LIN {X -0.071,Y -649.806,Z 548.445,A 0.000,B 0.000,C 90.000,E1 296.052} C_DIS
LIN {X 0.120,Y -649.563,Z 548.442,A 0.000,B 0.000,C 90.000,E1 295.540} C_DIS
LIN {X 0.217,Y -649.367,Z 548.441,A 0.000,B 0.000,C 90.000,E1 295.283} C_DIS
LIN {X -0.141,Y -646.576,Z 548.437,A 0.000,B 0.000,C 90.000,E1 294.695} C_DIS
LIN {X -0.098,Y -645.526,Z 548.436,A 0.000,B 0.000,C 90.000,E1 294.567} C_DIS
LIN {X -0.323,Y -643.886,Z 548.436,A 0.000,B 0.000,C 90.000,E1 294.463} C_DIS
LIN {X -0.018,Y -639.889,Z 548.434,A 0.000,B 0.000,C 90.000,E1 294.079} C_DIS
LIN {X 0.281,Y -635.567,Z 548.433,A 0.000,B 0.000,C 90.000,E1 293.823} C_DIS
LIN {X -0.032,Y -633.990,Z 548.432,A 0.000,B 0.000,C 90.000,E1 293.770} C_DIS
LIN {X -0.087,Y -632.744,Z 548.432,A 0.000,B 0.000,C 90.000,E1 293.695} C_DIS
LIN {X -0.057,Y -629.987,Z 548.431,A 0.000,B 0.000,C 90.000,E1 293.567} C_DIS
LIN {X -0.135,Y -626.756,Z 548.430,A 0.000,B 0.000,C 90.000,E1 293.462} C_DIS
LIN {X 0.125,Y -623.496,Z 548.429,A 0.000,B 0.000,C 90.000,E1 293.259} C_DIS
LIN {X 0.359,Y -616.119,Z 548.428,A 0.000,B 0.000,C 90.000,E1 292.950} C_DIS
LIN {X -0.008,Y -600.900,Z 548.425,A 0.000,B 0.000,C 90.000,E1 292.461} C_DIS
LIN {X -0.245,Y -582.055,Z 548.421,A 0.000,B 0.000,C 90.000,E1 291.844} C_DIS
LIN {X -0.113,Y -580.503,Z 548.421,A 0.000,B 0.000,C 90.000,E1 291.770} C_DIS
LIN {X 0.230,Y -574.157,Z 548.419,A 0.000,B 0.000,C 90.000,E1 291.408} C_DIS
LIN {X 0.077,Y -570.935,Z 548.418,A 0.000,B 0.000,C 90.000,E1 291.173} C_DIS
LIN {X -0.014,Y -570.080,Z 548.417,A 0.000,B 0.000,C 90.000,E1 291.046} C_DIS
LIN {X -0.057,Y -570.072,Z 548.417,A 0.000,B 0.000,C 90.000,E1 291.046} C_DIS
LIN {X 0.228,Y -569.535,Z 548.414,A 0.000,B 0.000,C 90.000,E1 290.556} C_DIS
LIN {X -0.116,Y -569.520,Z 548.405,A 0.000,B 0.000,C 90.000,E1 288.960} C_DIS
LIN {X -0.023,Y -569.321,Z 548.398,A 0.000,B 0.000,C 90.000,E1 287.583} C_DIS
LIN {X -0.099,Y -569.023,Z 548.392,A 0.000,B 0.000,C 90.000,E1 286.496} C_DIS
LIN {X 0.205,Y -568.590,Z 548.386,A 0.000,B 0.000,C 90.000,E1 285.371} C_DIS
LIN {X 0.131,Y -567.803,Z 548.378,A 0.000,B 0.000,C 90.000,E1 284.008} C_DIS
LIN {X 0.037,Y -567.041,Z 548.370,A 0.000,B 0.000,C 90.000,E1 282.647} C_DIS
LIN {X -0.030,Y -566.172,Z 548.361,A 0.000,B 0.000,C 90.000,E1 281.007} C_DIS
LIN {X -0.149,Y -565.171,Z 548.350,A 0.000,B 0.000,C 90.000,E1 279.095} C_DIS
LIN {X -0.281,Y -564.291,Z 548.340,A 0.000,B 0.000,C 90.000,E1 277.182} C_DIS
LIN {X -0.197,Y -563.753,Z 548.332,A 0.000,B 0.000,C 90.000,E1 275.796} C_DIS
LIN {X -0.082,Y -563.094,Z 548.323,A 0.000,B 0.000,C 90.000,E1 274.131} C_DIS
LIN {X -0.079,Y -562.422,Z 548.315,A 0.000,B 0.000,C 90.000,E1 272.751} C_DIS
LIN {X -0.026,Y -561.613,Z 548.306,A 0.000,B 0.000,C 90.000,E1 271.088} C_DIS
LIN {X 0.096,Y -560.451,Z 548.295,A 0.000,B 0.000,C 90.000,E1 269.141} C_DIS
LIN {X 0.017,Y -559.633,Z 548.288,A 0.000,B 0.000,C 90.000,E1 267.764} C_DIS
LIN {X -0.073,Y -558.784,Z 548.280,A 0.000,B 0.000,C 90.000,E1 266.388} C_DIS
LIN {X 0.055,Y -557.518,Z 548.269,A 0.000,B 0.000,C 90.000,E1 264.432} C_DIS
LIN {X 0.083,Y -556.351,Z 548.260,A 0.000,B 0.000,C 90.000,E1 262.761} C_DIS
LIN {X 0.022,Y -555.263,Z 548.252,A 0.000,B 0.000,C 90.000,E1 261.376} C_DIS
LIN {X -0.141,Y -554.368,Z 548.247,A 0.000,B 0.000,C 90.000,E1 260.557} C_DIS
LIN {X 0.209,Y -551.666,Z 548.235,A 0.000,B 0.000,C 90.000,E1 258.285} C_DIS
LIN {X 0.246,Y -550.027,Z 548.227,A 0.000,B 0.000,C 90.000,E1 256.881} C_DIS
LIN {X -0.156,Y -548.168,Z 548.219,A 0.000,B 0.000,C 90.000,E1 255.519} C_DIS
LIN {X -0.153,Y -546.644,Z 548.213,A 0.000,B 0.000,C 90.000,E1 254.393} C_DIS
LIN {X -0.176,Y -544.912,Z 548.207,A 0.000,B 0.000,C 90.000,E1 253.268} C_DIS
LIN {X -0.291,Y -542.060,Z 548.198,A 0.000,B 0.000,C 90.000,E1 251.583} C_DIS
LIN {X -0.054,Y -540.059,Z 548.191,A 0.000,B 0.000,C 90.000,E1 250.423} C_DIS
LIN {X -0.066,Y -538.426,Z 548.187,A 0.000,B 0.000,C 90.000,E1 249.571} C_DIS
LIN {X -0.167,Y -535.507,Z 548.179,A 0.000,B 0.000,C 90.000,E1 248.156} C_DIS
LIN {X -0.114,Y -532.460,Z 548.171,A 0.000,B 0.000,C 90.000,E1 246.719} C_DIS
LIN {X -0.115,Y -529.083,Z 548.163,A 0.000,B 0.000,C 90.000,E1 245.281} C_DIS
LIN {X 0.113,Y -526.222,Z 548.156,A 0.000,B 0.000,C 90.000,E1 244.101} C_DIS
LIN {X 0.047,Y -523.179,Z 548.150,A 0.000,B 0.000,C 90.000,E1 242.948} C_DIS
LIN {X -0.145,Y -519.278,Z 548.142,A 0.000,B 0.000,C 90.000,E1 241.513} C_DIS
LIN {X 0.298,Y -515.279,Z 548.134,A 0.000,B 0.000,C 90.000,E1 239.999} C_DIS
LIN {X -0.037,Y -512.768,Z 548.129,A 0.000,B 0.000,C 90.000,E1 239.154} C_DIS
LIN {X 0.101,Y -508.301,Z 548.120,A 0.000,B 0.000,C 90.000,E1 237.661} C_DIS
LIN {X 0.156,Y -503.856,Z 548.112,A 0.000,B 0.000,C 90.000,E1 236.167} C_DIS
LIN {X 0.151,Y -497.818,Z 548.101,A 0.000,B 0.000,C 90.000,E1 234.069} C_DIS
LIN {X -0.113,Y -492.012,Z 548.089,A 0.000,B 0.000,C 90.000,E1 231.984} C_DIS
LIN {X -0.087,Y -485.498,Z 548.075,A 0.000,B 0.000,C 90.000,E1 229.542} C_DIS
LIN {X 0.088,Y -480.746,Z 548.065,A 0.000,B 0.000,C 90.000,E1 227.676} C_DIS
LIN {X 0.266,Y -475.303,Z 548.053,A 0.000,B 0.000,C 90.000,E1 225.486} C_DIS
LIN {X -0.044,Y -470.062,Z 548.041,A 0.000,B 0.000,C 90.000,E1 223.338} C_DIS
LIN {X 0.098,Y -465.668,Z 548.030,A 0.000,B 0.000,C 90.000,E1 221.434} C_DIS
LIN {X 0.069,Y -462.782,Z 548.023,A 0.000,B 0.000,C 90.000,E1 220.172} C_DIS
LIN {X 0.133,Y -458.572,Z 548.013,A 0.000,B 0.000,C 90.000,E1 218.257} C_DIS
LIN {X -0.181,Y -454.400,Z 548.002,A 0.000,B 0.000,C 90.000,E1 216.377} C_DIS
LIN {X -0.153,Y -449.717,Z 547.990,A 0.000,B 0.000,C 90.000,E1 214.119} C_DIS
LIN {X 0.166,Y -445.819,Z 547.979,A 0.000,B 0.000,C 90.000,E1 212.133} C_DIS
LIN {X 0.028,Y -440.845,Z 547.964,A 0.000,B 0.000,C 90.000,E1 209.539} C_DIS
LIN {X -0.014,Y -438.499,Z 547.957,A 0.000,B 0.000,C 90.000,E1 208.231} C_DIS
LIN {X -0.039,Y -434.540,Z 547.944,A 0.000,B 0.000,C 90.000,E1 205.924} C_DIS
LIN {X 0.037,Y -430.766,Z 547.931,A 0.000,B 0.000,C 90.000,E1 203.590} C_DIS
LIN {X 0.220,Y -428.218,Z 547.922,A 0.000,B 0.000,C 90.000,E1 201.897} C_DIS
LIN {X 0.005,Y -424.041,Z 547.905,A 0.000,B 0.000,C 90.000,E1 198.906} C_DIS
LIN {X 0.005,Y -420.535,Z 547.890,A 0.000,B 0.000,C 90.000,E1 196.205} C_DIS
LIN {X 0.020,Y -417.754,Z 547.877,A 0.000,B 0.000,C 90.000,E1 193.828} C_DIS
LIN {X -0.077,Y -415.924,Z 547.869,A 0.000,B 0.000,C 90.000,E1 192.479} C_DIS
LIN {X -0.034,Y -413.303,Z 547.858,A 0.000,B 0.000,C 90.000,E1 190.423} C_DIS
LIN {X 0.190,Y -410.163,Z 547.843,A 0.000,B 0.000,C 90.000,E1 187.644} C_DIS
LIN {X -0.181,Y -407.426,Z 547.827,A 0.000,B 0.000,C 90.000,E1 184.935} C_DIS
LIN {X 0.110,Y -404.964,Z 547.812,A 0.000,B 0.000,C 90.000,E1 182.121} C_DIS
LIN {X -0.086,Y -403.054,Z 547.798,A 0.000,B 0.000,C 90.000,E1 179.714} C_DIS
LIN {X 0.111,Y -401.910,Z 547.787,A 0.000,B 0.000,C 90.000,E1 177.593} C_DIS
LIN {X -0.121,Y -400.938,Z 547.773,A 0.000,B 0.000,C 90.000,E1 175.179} C_DIS
LIN {X 0.067,Y -400.447,Z 547.762,A 0.000,B 0.000,C 90.000,E1 173.053} C_DIS
LIN {X -0.095,Y -400.252,Z 547.746,A 0.000,B 0.000,C 90.000,E1 170.274} C_DIS
LIN {X -0.032,Y -400.353,Z 547.732,A 0.000,B 0.000,C 90.000,E1 167.813} C_DIS
LIN {X 0.115,Y -400.928,Z 547.717,A 0.000,B 0.000,C 90.000,E1 164.991} C_DIS
LIN {X 0.022,Y -401.592,Z 547.705,A 0.000,B 0.000,C 90.000,E1 162.906} C_DIS
LIN {X -0.098,Y -402.599,Z 547.692,A 0.000,B 0.000,C 90.000,E1 160.477} C_DIS
LIN {X -0.098,Y -403.321,Z 547.684,A 0.000,B 0.000,C 90.000,E1 159.082} C_DIS
LIN {X 0.117,Y -404.689,Z 547.670,A 0.000,B 0.000,C 90.000,E1 156.613} C_DIS
LIN {X 0.058,Y -405.995,Z 547.659,A 0.000,B 0.000,C 90.000,E1 154.537} C_DIS
LIN {X -0.070,Y -407.105,Z 547.649,A 0.000,B 0.000,C 90.000,E1 152.820} C_DIS
LIN {X 0.202,Y -408.157,Z 547.639,A 0.000,B 0.000,C 90.000,E1 151.051} C_DIS
LIN {X 0.144,Y -409.138,Z 547.630,A 0.000,B 0.000,C 90.000,E1 149.331} C_DIS
LIN {X 0.238,Y -410.037,Z 547.618,A 0.000,B 0.000,C 90.000,E1 147.248} C_DIS
LIN {X 0.227,Y -410.762,Z 547.607,A 0.000,B 0.000,C 90.000,E1 145.182} C_DIS
LIN {X -0.033,Y -411.189,Z 547.597,A 0.000,B 0.000,C 90.000,E1 143.497} C_DIS
LIN {X -0.045,Y -411.527,Z 547.588,A 0.000,B 0.000,C 90.000,E1 141.778} C_DIS
LIN {X -0.022,Y -411.669,Z 547.580,A 0.000,B 0.000,C 90.000,E1 140.400} C_DIS
LIN {X -0.087,Y -411.745,Z 547.570,A 0.000,B 0.000,C 90.000,E1 138.690} C_DIS
LIN {X -0.033,Y -411.839,Z 547.559,A 0.000,B 0.000,C 90.000,E1 136.620} C_DIS
LIN {X 0.146,Y -411.978,Z 547.546,A 0.000,B 0.000,C 90.000,E1 134.190} C_DIS
LIN {X -0.096,Y -412.097,Z 547.534,A 0.000,B 0.000,C 90.000,E1 132.162} C_DIS
LIN {X -0.052,Y -412.028,Z 547.527,A 0.000,B 0.000,C 90.000,E1 130.782} C_DIS
LIN {X 0.135,Y -411.889,Z 547.521,A 0.000,B 0.000,C 90.000,E1 129.725} C_DIS
LIN {X 0.058,Y -411.552,Z 547.515,A 0.000,B 0.000,C 90.000,E1 128.705} C_DIS
LIN {X -0.101,Y -410.959,Z 547.508,A 0.000,B 0.000,C 90.000,E1 127.523} C_DIS
LIN {X -0.139,Y -410.959,Z 547.508,A 0.000,B 0.000,C 90.000,E1 127.523} C_DIS
LIN {X -0.009,Y -415.555,Z 547.500,A 0.000,B 0.000,C 90.000,E1 125.964} C_DIS
LIN {X 0.075,Y -425.946,Z 547.477,A 0.000,B 0.000,C 90.000,E1 121.878} C_DIS
LIN {X 0.029,Y -430.952,Z 547.468,A 0.000,B 0.000,C 90.000,E1 120.207} C_DIS
LIN {X -0.022,Y -440.011,Z 547.448,A 0.000,B 0.000,C 90.000,E1 116.565} C_DIS
LIN {X 0.211,Y -444.409,Z 547.439,A 0.000,B 0.000,C 90.000,E1 115.027} C_DIS
LIN {X 0.170,Y -444.437,Z 547.439,A 0.000,B 0.000,C 90.000,E1 115.027} C_DIS
LIN {X -0.031,Y -463.005,Z 547.435,A 0.000,B 0.000,C 90.000,E1 114.259} C_DIS
LIN {X -0.080,Y -482.164,Z 547.430,A 0.000,B 0.000,C 90.000,E1 113.462} C_DIS
LIN {X 0.029,Y -488.924,Z 547.429,A 0.000,B 0.000,C 90.000,E1 113.153} C_DIS
LIN {X 0.224,Y -495.886,Z 547.427,A 0.000,B 0.000,C 90.000,E1 112.823} C_DIS
LIN {X 0.092,Y -509.292,Z 547.423,A 0.000,B 0.000,C 90.000,E1 112.206} C_DIS
LIN {X -0.001,Y -515.930,Z 547.422,A 0.000,B 0.000,C 90.000,E1 111.897} C_DIS
LIN {X -0.195,Y -522.483,Z 547.420,A 0.000,B 0.000,C 90.000,E1 111.589} C_DIS
LIN {X -0.142,Y -533.967,Z 547.417,A 0.000,B 0.000,C 90.000,E1 110.972} C_DIS
LIN {X -0.109,Y -540.286,Z 547.414,A 0.000,B 0.000,C 90.000,E1 110.610} C_DIS
LIN {X -0.020,Y -547.960,Z 547.412,A 0.000,B 0.000,C 90.000,E1 110.120} C_DIS
LIN {X -0.009,Y -553.960,Z 547.409,A 0.000,B 0.000,C 90.000,E1 109.704} C_DIS
LIN {X -0.265,Y -558.363,Z 547.408,A 0.000,B 0.000,C 90.000,E1 109.396} C_DIS
LIN {X -0.077,Y -563.993,Z 547.405,A 0.000,B 0.000,C 90.000,E1 108.906} C_DIS
LIN {X -0.013,Y -570.154,Z 547.402,A 0.000,B 0.000,C 90.000,E1 108.308} C_DIS
LIN {X 0.142,Y -574.689,Z 547.399,A 0.000,B 0.000,C 90.000,E1 107.819} C_DIS
LIN {X -0.199,Y -577.977,Z 547.397,A 0.000,B 0.000,C 90.000,E1 107.457} C_DIS
LIN {X 0.001,Y -580.308,Z 547.395,A 0.000,B 0.000,C 90.000,E1 107.166} C_DIS
LIN {X 0.297,Y -585.084,Z 547.392,A 0.000,B 0.000,C 90.000,E1 106.496} C_DIS
LIN {X 0.128,Y -589.806,Z 547.388,A 0.000,B 0.000,C 90.000,E1 105.843} C_DIS
LIN {X -0.079,Y -594.976,Z 547.384,A 0.000,B 0.000,C 90.000,E1 105.064} C_DIS
LIN {X -0.099,Y -598.175,Z 547.381,A 0.000,B 0.000,C 90.000,E1 104.537} C_DIS
LIN {X 0.210,Y -602.588,Z 547.376,A 0.000,B 0.000,C 90.000,E1 103.716} C_DIS
LIN {X 0.250,Y -609.039,Z 547.370,A 0.000,B 0.000,C 90.000,E1 102.535} C_DIS
LIN {X 0.085,Y -613.063,Z 547.365,A 0.000,B 0.000,C 90.000,E1 101.771} C_DIS
LIN {X 0.194,Y -615.665,Z 547.363,A 0.000,B 0.000,C 90.000,E1 101.243} C_DIS
LIN {X -0.032,Y -619.092,Z 547.358,A 0.000,B 0.000,C 90.000,E1 100.489} C_DIS
LIN {X -0.117,Y -622.267,Z 547.354,A 0.000,B 0.000,C 90.000,E1 99.726} C_DIS
LIN {X 0.211,Y -628.750,Z 547.346,A 0.000,B 0.000,C 90.000,E1 98.163} C_DIS
LIN {X -0.174,Y -632.914,Z 547.340,A 0.000,B 0.000,C 90.000,E1 97.182} C_DIS
LIN {X -0.071,Y -637.945,Z 547.333,A 0.000,B 0.000,C 90.000,E1 95.910} C_DIS
LIN {X 0.236,Y -641.480,Z 547.327,A 0.000,B 0.000,C 90.000,E1 94.878} C_DIS
LIN {X 0.200,Y -643.859,Z 547.323,A 0.000,B 0.000,C 90.000,E1 94.131} C_DIS
LIN {X -0.044,Y -646.678,Z 547.318,A 0.000,B 0.000,C 90.000,E1 93.154} C_DIS
LIN {X -0.034,Y -648.534,Z 547.313,A 0.000,B 0.000,C 90.000,E1 92.407} C_DIS
LIN {X -0.014,Y -649.948,Z 547.309,A 0.000,B 0.000,C 90.000,E1 91.661} C_DIS
LIN {X 0.000,Y -651.078,Z 547.305,A 0.000,B 0.000,C 90.000,E1 90.917} C_DIS
LIN {X 0.234,Y -651.671,Z 547.302,A 0.000,B 0.000,C 90.000,E1 90.401} C_DIS
LIN {X 0.270,Y -652.305,Z 547.298,A 0.000,B 0.000,C 90.000,E1 89.656} C_DIS
LIN {X 0.309,Y -652.508,Z 547.294,A 0.000,B 0.000,C 90.000,E1 88.912} C_DIS
LIN {X -0.100,Y -652.546,Z 547.291,A 0.000,B 0.000,C 90.000,E1 88.453} C_DIS
LIN {X -0.040,Y -652.236,Z 547.287,A 0.000,B 0.000,C 90.000,E1 87.707} C_DIS
LIN {X -0.009,Y -651.640,Z 547.283,A 0.000,B 0.000,C 90.000,E1 86.963} C_DIS
LIN {X 0.047,Y -650.882,Z 547.279,A 0.000,B 0.000,C 90.000,E1 86.216} C_DIS
LIN {X 0.097,Y -649.758,Z 547.275,A 0.000,B 0.000,C 90.000,E1 85.469} C_DIS
LIN {X -0.029,Y -648.010,Z 547.269,A 0.000,B 0.000,C 90.000,E1 84.489} C_DIS
LIN {X 0.159,Y -647.012,Z 547.267,A 0.000,B 0.000,C 90.000,E1 83.976} C_DIS
LIN {X 0.235,Y -645.175,Z 547.263,A 0.000,B 0.000,C 90.000,E1 83.223} C_DIS
LIN {X 0.302,Y -643.082,Z 547.258,A 0.000,B 0.000,C 90.000,E1 82.470} C_DIS
LIN {X 0.091,Y -639.999,Z 547.253,A 0.000,B 0.000,C 90.000,E1 81.489} C_DIS
LIN {X 0.281,Y -638.350,Z 547.250,A 0.000,B 0.000,C 90.000,E1 80.971} C_DIS
LIN {X 0.097,Y -634.711,Z 547.244,A 0.000,B 0.000,C 90.000,E1 79.982} C_DIS
LIN {X -0.134,Y -630.688,Z 547.239,A 0.000,B 0.000,C 90.000,E1 78.993} C_DIS
LIN {X -0.292,Y -626.257,Z 547.233,A 0.000,B 0.000,C 90.000,E1 77.993} C_DIS
LIN {X 0.106,Y -621.422,Z 547.228,A 0.000,B 0.000,C 90.000,E1 76.937} C_DIS
LIN {X 0.273,Y -618.808,Z 547.225,A 0.000,B 0.000,C 90.000,E1 76.408} C_DIS
LIN {X -0.218,Y -615.267,Z 547.221,A 0.000,B 0.000,C 90.000,E1 75.811} C_DIS
LIN {X -0.290,Y -611.517,Z 547.218,A 0.000,B 0.000,C 90.000,E1 75.172} C_DIS
LIN {X -0.245,Y -607.412,Z 547.214,A 0.000,B 0.000,C 90.000,E1 74.519} C_DIS
LIN {X -0.235,Y -602.951,Z 547.210,A 0.000,B 0.000,C 90.000,E1 73.866} C_DIS
LIN {X -0.094,Y -598.067,Z 547.207,A 0.000,B 0.000,C 90.000,E1 73.196} C_DIS
LIN {X 0.132,Y -594.633,Z 547.204,A 0.000,B 0.000,C 90.000,E1 72.779} C_DIS
LIN {X -0.226,Y -592.933,Z 547.203,A 0.000,B 0.000,C 90.000,E1 72.598} C_DIS
LIN {X -0.060,Y -588.167,Z 547.200,A 0.000,B 0.000,C 90.000,E1 72.054} C_DIS
LIN {X 0.188,Y -583.017,Z 547.197,A 0.000,B 0.000,C 90.000,E1 71.511} C_DIS
LIN {X -0.070,Y -580.127,Z 547.196,A 0.000,B 0.000,C 90.000,E1 71.275} C_DIS
LIN {X 0.274,Y -576.665,Z 547.194,A 0.000,B 0.000,C 90.000,E1 70.913} C_DIS
LIN {X -0.110,Y -571.441,Z 547.192,A 0.000,B 0.000,C 90.000,E1 70.496} C_DIS
LIN {X -0.117,Y -565.989,Z 547.189,A 0.000,B 0.000,C 90.000,E1 70.061} C_DIS
LIN {X -0.106,Y -561.746,Z 547.188,A 0.000,B 0.000,C 90.000,E1 69.752} C_DIS
LIN {X 0.092,Y -555.767,Z 547.185,A 0.000,B 0.000,C 90.000,E1 69.337} C_DIS
LIN {X -0.024,Y -548.840,Z 547.183,A 0.000,B 0.000,C 90.000,E1 68.954} C_DIS
LIN {X 0.168,Y -543.961,Z 547.182,A 0.000,B 0.000,C 90.000,E1 68.666} C_DIS
LIN {X 0.158,Y -536.911,Z 547.180,A 0.000,B 0.000,C 90.000,E1 68.337} C_DIS
LIN {X 0.211,Y -531.587,Z 547.179,A 0.000,B 0.000,C 90.000,E1 68.103} C_DIS
LIN {X -0.037,Y -520.907,Z 547.176,A 0.000,B 0.000,C 90.000,E1 67.720} C_DIS
LIN {X -0.262,Y -513.715,Z 547.175,A 0.000,B 0.000,C 90.000,E1 67.486} C_DIS
LIN {X 0.008,Y -502.871,Z 547.173,A 0.000,B 0.000,C 90.000,E1 67.102} C_DIS
LIN {X -0.116,Y -488.459,Z 547.170,A 0.000,B 0.000,C 90.000,E1 66.666} C_DIS
LIN {X 0.228,Y -462.841,Z 547.166,A 0.000,B 0.000,C 90.000,E1 65.793} C_DIS
LIN {X 0.197,Y -462.827,Z 547.166,A 0.000,B 0.000,C 90.000,E1 65.793} C_DIS
LIN {X 0.180,Y -455.513,Z 547.144,A 0.000,B 0.000,C 90.000,E1 61.897} C_DIS
LIN {X 0.185,Y -445.565,Z 547.119,A 0.000,B 0.000,C 90.000,E1 57.375} C_DIS
LIN {X 0.001,Y -443.781,Z 547.114,A 0.000,B 0.000,C 90.000,E1 56.421} C_DIS
LIN {X -0.160,Y -441.605,Z 547.109,A 0.000,B 0.000,C 90.000,E1 55.595} C_DIS
LIN {X -0.200,Y -441.599,Z 547.109,A 0.000,B 0.000,C 90.000,E1 55.595} C_DIS
LIN {X 0.118,Y -444.210,Z 547.101,A 0.000,B 0.000,C 90.000,E1 54.116} C_DIS
LIN {X -0.138,Y -446.445,Z 547.094,A 0.000,B 0.000,C 90.000,E1 52.844} C_DIS
LIN {X 0.236,Y -449.164,Z 547.084,A 0.000,B 0.000,C 90.000,E1 51.170} C_DIS
LIN {X -0.028,Y -451.203,Z 547.077,A 0.000,B 0.000,C 90.000,E1 49.908} C_DIS
LIN {X -0.259,Y -453.562,Z 547.068,A 0.000,B 0.000,C 90.000,E1 48.324} C_DIS
LIN {X 0.142,Y -455.309,Z 547.061,A 0.000,B 0.000,C 90.000,E1 46.986} C_DIS
LIN {X -0.099,Y -456.400,Z 547.056,A 0.000,B 0.000,C 90.000,E1 46.053} C_DIS
LIN {X -0.011,Y -457.296,Z 547.050,A 0.000,B 0.000,C 90.000,E1 45.081} C_DIS
LIN {X 0.122,Y -458.195,Z 547.043,A 0.000,B 0.000,C 90.000,E1 43.785} C_DIS
LIN {X -0.124,Y -458.624,Z 547.040,A 0.000,B 0.000,C 90.000,E1 43.176} C_DIS
LIN {X 0.019,Y -459.133,Z 547.033,A 0.000,B 0.000,C 90.000,E1 41.881} C_DIS
LIN {X -0.107,Y -459.395,Z 547.026,A 0.000,B 0.000,C 90.000,E1 40.620} C_DIS
LIN {X 0.071,Y -459.405,Z 547.019,A 0.000,B 0.000,C 90.000,E1 39.322} C_DIS
LIN {X 0.050,Y -459.237,Z 547.010,A 0.000,B 0.000,C 90.000,E1 37.729} C_DIS
LIN {X 0.131,Y -458.642,Z 546.999,A 0.000,B 0.000,C 90.000,E1 35.804} C_DIS
LIN {X -0.070,Y -457.878,Z 546.988,A 0.000,B 0.000,C 90.000,E1 33.913} C_DIS
LIN {X -0.053,Y -456.995,Z 546.976,A 0.000,B 0.000,C 90.000,E1 31.671} C_DIS
LIN {X -0.015,Y -456.257,Z 546.965,A 0.000,B 0.000,C 90.000,E1 29.745} C_DIS
LIN {X -0.116,Y -455.310,Z 546.953,A 0.000,B 0.000,C 90.000,E1 27.513} C_DIS
LIN {X -0.047,Y -454.682,Z 546.944,A 0.000,B 0.000,C 90.000,E1 25.899} C_DIS
LIN {X -0.098,Y -453.829,Z 546.930,A 0.000,B 0.000,C 90.000,E1 23.334} C_DIS
LIN {X 0.184,Y -453.283,Z 546.917,A 0.000,B 0.000,C 90.000,E1 21.046} C_DIS
LIN {X 0.025,Y -452.802,Z 546.903,A 0.000,B 0.000,C 90.000,E1 18.489} C_DIS
LIN {X 0.129,Y -452.720,Z 546.888,A 0.000,B 0.000,C 90.000,E1 15.898} C_DIS
LIN {X -0.083,Y -453.063,Z 546.871,A 0.000,B 0.000,C 90.000,E1 12.703} C_DIS
LIN {X -0.217,Y -454.109,Z 546.853,A 0.000,B 0.000,C 90.000,E1 9.500} C_DIS
LIN {X -0.203,Y -455.563,Z 546.837,A 0.000,B 0.000,C 90.000,E1 6.606} C_DIS
LIN {X 0.025,Y -457.200,Z 546.822,A 0.000,B 0.000,C 90.000,E1 4.012} C_DIS
LIN {X 0.201,Y -459.229,Z 546.808,A 0.000,B 0.000,C 90.000,E1 1.432} C_DIS
LIN {X 0.123,Y -461.568,Z 546.795,A 0.000,B 0.000,C 90.000,E1 359.141} C_DIS
LIN {X 0.004,Y -463.826,Z 546.785,A 0.000,B 0.000,C 90.000,E1 357.249} C_DIS
LIN {X 0.214,Y -466.774,Z 546.772,A 0.000,B 0.000,C 90.000,E1 355.008} C_DIS
LIN {X -0.216,Y -468.484,Z 546.765,A 0.000,B 0.000,C 90.000,E1 353.799} C_DIS
LIN {X -0.066,Y -471.004,Z 546.755,A 0.000,B 0.000,C 90.000,E1 351.894} C_DIS
LIN {X 0.168,Y -474.973,Z 546.739,A 0.000,B 0.000,C 90.000,E1 349.050} C_DIS
LIN {X 0.087,Y -478.476,Z 546.727,A 0.000,B 0.000,C 90.000,E1 346.881} C_DIS
LIN {X -0.260,Y -482.194,Z 546.715,A 0.000,B 0.000,C 90.000,E1 344.755} C_DIS
LIN {X 0.083,Y -487.370,Z 546.700,A 0.000,B 0.000,C 90.000,E1 341.945} C_DIS
LIN {X 0.053,Y -490.959,Z 546.690,A 0.000,B 0.000,C 90.000,E1 340.115} C_DIS
LIN {X 0.155,Y -495.167,Z 546.678,A 0.000,B 0.000,C 90.000,E1 337.975} C_DIS
LIN {X 0.019,Y -498.611,Z 546.668,A 0.000,B 0.000,C 90.000,E1 336.177} C_DIS
LIN {X 0.086,Y -501.355,Z 546.659,A 0.000,B 0.000,C 90.000,E1 334.665} C_DIS
LIN {X 0.047,Y -504.590,Z 546.649,A 0.000,B 0.000,C 90.000,E1 332.871} C_DIS
LIN {X -0.079,Y -506.718,Z 546.643,A 0.000,B 0.000,C 90.000,E1 331.691} C_DIS
LIN {X -0.129,Y -510.331,Z 546.631,A 0.000,B 0.000,C 90.000,E1 329.616} C_DIS
LIN {X -0.009,Y -512.971,Z 546.623,A 0.000,B 0.000,C 90.000,E1 328.122} C_DIS
LIN {X -0.264,Y -516.678,Z 546.612,A 0.000,B 0.000,C 90.000,E1 326.087} C_DIS
LIN {X 0.204,Y -519.846,Z 546.602,A 0.000,B 0.000,C 90.000,E1 324.276} C_DIS
LIN {X -0.100,Y -522.978,Z 546.592,A 0.000,B 0.000,C 90.000,E1 322.557} C_DIS
LIN {X -0.050,Y -526.825,Z 546.581,A 0.000,B 0.000,C 90.000,E1 320.517} C_DIS
LIN {X 0.025,Y -530.937,Z 546.569,A 0.000,B 0.000,C 90.000,E1 318.485} C_DIS
LIN {X -0.240,Y -536.135,Z 546.557,A 0.000,B 0.000,C 90.000,E1 316.215} C_DIS
LIN {X 0.019,Y -543.111,Z 546.541,A 0.000,B 0.000,C 90.000,E1 313.338} C_DIS
LIN {X 0.058,Y -546.696,Z 546.533,A 0.000,B 0.000,C 90.000,E1 311.919} C_DIS
LIN {X -0.164,Y -550.764,Z 546.524,A 0.000,B 0.000,C 90.000,E1 310.253} C_DIS
LIN {X 0.299,Y -552.109,Z 546.520,A 0.000,B 0.000,C 90.000,E1 309.644} C_DIS
LIN {X 0.057,Y -554.366,Z 546.516,A 0.000,B 0.000,C 90.000,E1 308.830} C_DIS
LIN {X 0.125,Y -555.260,Z 546.514,A 0.000,B 0.000,C 90.000,E1 308.543} C_DIS
LIN {X 0.198,Y -556.794,Z 546.513,A 0.000,B 0.000,C 90.000,E1 308.257} C_DIS
LIN {X -0.163,Y -558.016,Z 546.511,A 0.000,B 0.000,C 90.000,E1 308.016} C_DIS
LIN {X -0.207,Y -560.843,Z 546.509,A 0.000,B 0.000,C 90.000,E1 307.604} C_DIS
LIN {X 0.009,Y -561.739,Z 546.508,A 0.000,B 0.000,C 90.000,E1 307.443} C_DIS
LIN {X 0.086,Y -565.665,Z 546.506,A 0.000,B 0.000,C 90.000,E1 306.996} C_DIS
LIN {X 0.074,Y -577.991,Z 546.500,A 0.000,B 0.000,C 90.000,E1 305.931} C_DIS
LIN {X 0.214,Y -584.483,Z 546.496,A 0.000,B 0.000,C 90.000,E1 305.311} C_DIS
LIN {X 0.122,Y -588.314,Z 546.494,A 0.000,B 0.000,C 90.000,E1 304.945} C_DIS
LIN {X -0.173,Y -594.560,Z 546.491,A 0.000,B 0.000,C 90.000,E1 304.326} C_DIS
LIN {X 0.013,Y -600.747,Z 546.487,A 0.000,B 0.000,C 90.000,E1 303.658} C_DIS
LIN {X -0.136,Y -610.259,Z 546.481,A 0.000,B 0.000,C 90.000,E1 302.625} C_DIS
LIN {X 0.375,Y -617.069,Z 546.477,A 0.000,B 0.000,C 90.000,E1 301.799} C_DIS
LIN {X 0.102,Y -624.754,Z 546.472,A 0.000,B 0.000,C 90.000,E1 300.924} C_DIS
LIN {X 0.115,Y -629.586,Z 546.468,A 0.000,B 0.000,C 90.000,E1 300.285} C_DIS
LIN {X -0.071,Y -633.038,Z 546.466,A 0.000,B 0.000,C 90.000,E1 299.795} C_DIS
LIN {X 0.019,Y -636.516,Z 546.462,A 0.000,B 0.000,C 90.000,E1 299.155} C_DIS
LIN {X -0.113,Y -639.427,Z 546.459,A 0.000,B 0.000,C 90.000,E1 298.537} C_DIS
LIN {X 0.126,Y -642.898,Z 546.453,A 0.000,B 0.000,C 90.000,E1 297.513} C_DIS
LIN {X 0.267,Y -644.533,Z 546.450,A 0.000,B 0.000,C 90.000,E1 297.001} C_DIS
LIN {X -0.158,Y -645.835,Z 546.447,A 0.000,B 0.000,C 90.000,E1 296.539} C_DIS
LIN {X -0.080,Y -646.463,Z 546.446,A 0.000,B 0.000,C 90.000,E1 296.283} C_DIS
LIN {X 0.002,Y -646.755,Z 546.445,A 0.000,B 0.000,C 90.000,E1 296.027} C_DIS
LIN {X -0.111,Y -646.598,Z 546.442,A 0.000,B 0.000,C 90.000,E1 295.540} C_DIS
LIN {X -0.026,Y -646.074,Z 546.440,A 0.000,B 0.000,C 90.000,E1 295.283} C_DIS
LIN {X 0.140,Y -644.044,Z 546.438,A 0.000,B 0.000,C 90.000,E1 294.771} C_DIS
LIN {X 0.251,Y -640.832,Z 546.436,A 0.000,B 0.000,C 90.000,E1 294.387} C_DIS
LIN {X 0.065,Y -638.226,Z 546.434,A 0.000,B 0.000,C 90.000,E1 294.155} C_DIS
LIN {X 0.108,Y -635.689,Z 546.434,A 0.000,B 0.000,C 90.000,E1 294.027} C_DIS
LIN {X -0.231,Y -632.967,Z 546.433,A 0.000,B 0.000,C 90.000,E1 293.898} C_DIS
LIN {X 0.102,Y -632.502,Z 546.432,A 0.000,B 0.000,C 90.000,E1 293.823} C_DIS
LIN {X 0.160,Y -630.798,Z 546.432,A 0.000,B 0.000,C 90.000,E1 293.695} C_DIS
LIN {X -0.034,Y -627.696,Z 546.431,A 0.000,B 0.000,C 90.000,E1 293.590} C_DIS
LIN {X -0.110,Y -624.102,Z 546.430,A 0.000,B 0.000,C 90.000,E1 293.387} C_DIS
LIN {X 0.297,Y -622.357,Z 546.429,A 0.000,B 0.000,C 90.000,E1 293.259} C_DIS
LIN {X 0.242,Y -612.951,Z 546.427,A 0.000,B 0.000,C 90.000,E1 292.898} C_DIS
LIN {X 0.273,Y -600.603,Z 546.425,A 0.000,B 0.000,C 90.000,E1 292.461} C_DIS
LIN {X -0.003,Y -581.868,Z 546.421,A 0.000,B 0.000,C 90.000,E1 291.844} C_DIS
LIN {X 0.094,Y -576.724,Z 546.420,A 0.000,B 0.000,C 90.000,E1 291.589} C_DIS
LIN {X -0.191,Y -575.181,Z 546.420,A 0.000,B 0.000,C 90.000,E1 291.535} C_DIS
LIN {X 0.229,Y -571.555,Z 546.418,A 0.000,B 0.000,C 90.000,E1 291.227} C_DIS
LIN {X -0.202,Y -571.095,Z 546.418,A 0.000,B 0.000,C 90.000,E1 291.227} C_DIS
LIN {X -0.222,Y -570.643,Z 546.417,A 0.000,B 0.000,C 90.000,E1 291.099} C_DIS
LIN {X -0.252,Y -570.029,Z 546.414,A 0.000,B 0.000,C 90.000,E1 290.556} C_DIS
LIN {X 0.224,Y -570.059,Z 546.406,A 0.000,B 0.000,C 90.000,E1 289.141} C_DIS
LIN {X -0.217,Y -569.904,Z 546.399,A 0.000,B 0.000,C 90.000,E1 287.819} C_DIS
LIN {X -0.114,Y -569.570,Z 546.391,A 0.000,B 0.000,C 90.000,E1 286.441} C_DIS
LIN {X 0.202,Y -569.142,Z 546.385,A 0.000,B 0.000,C 90.000,E1 285.315} C_DIS
LIN {X -0.097,Y -568.179,Z 546.376,A 0.000,B 0.000,C 90.000,E1 283.703} C_DIS
LIN {X 0.059,Y -567.594,Z 546.370,A 0.000,B 0.000,C 90.000,E1 282.591} C_DIS
LIN {X -0.167,Y -566.890,Z 546.362,A 0.000,B 0.000,C 90.000,E1 281.243} C_DIS
LIN {X -0.131,Y -566.283,Z 546.356,A 0.000,B 0.000,C 90.000,E1 280.141} C_DIS
LIN {X 0.244,Y -565.481,Z 546.347,A 0.000,B 0.000,C 90.000,E1 278.454} C_DIS
LIN {X 0.043,Y -564.633,Z 546.336,A 0.000,B 0.000,C 90.000,E1 276.549} C_DIS
LIN {X 0.134,Y -564.109,Z 546.329,A 0.000,B 0.000,C 90.000,E1 275.163} C_DIS
LIN {X 0.154,Y -563.542,Z 546.321,A 0.000,B 0.000,C 90.000,E1 273.784} C_DIS
LIN {X -0.227,Y -562.558,Z 546.310,A 0.000,B 0.000,C 90.000,E1 271.892} C_DIS
LIN {X -0.267,Y -561.784,Z 546.303,A 0.000,B 0.000,C 90.000,E1 270.516} C_DIS
LIN {X -0.142,Y -560.628,Z 546.292,A 0.000,B 0.000,C 90.000,E1 268.568} C_DIS
LIN {X -0.132,Y -559.591,Z 546.283,A 0.000,B 0.000,C 90.000,E1 266.906} C_DIS
LIN {X 0.009,Y -558.286,Z 546.272,A 0.000,B 0.000,C 90.000,E1 264.951} C_DIS
LIN {X -0.143,Y -557.528,Z 546.266,A 0.000,B 0.000,C 90.000,E1 263.856} C_DIS
LIN {X -0.175,Y -556.555,Z 546.258,A 0.000,B 0.000,C 90.000,E1 262.470} C_DIS
LIN {X 0.190,Y -555.683,Z 546.252,A 0.000,B 0.000,C 90.000,E1 261.319} C_DIS
LIN {X 0.031,Y -554.773,Z 546.247,A 0.000,B 0.000,C 90.000,E1 260.500} C_DIS
LIN {X -0.153,Y -552.036,Z 546.235,A 0.000,B 0.000,C 90.000,E1 258.285} C_DIS
LIN {X -0.108,Y -550.358,Z 546.227,A 0.000,B 0.000,C 90.000,E1 256.881} C_DIS
LIN {X 0.027,Y -548.467,Z 546.219,A 0.000,B 0.000,C 90.000,E1 255.463} C_DIS
LIN {X 0.122,Y -546.498,Z 546.211,A 0.000,B 0.000,C 90.000,E1 254.047} C_DIS
LIN {X 0.245,Y -544.701,Z 546.205,A 0.000,B 0.000,C 90.000,E1 252.906} C_DIS
LIN {X 0.124,Y -541.782,Z 546.196,A 0.000,B 0.000,C 90.000,E1 251.221} C_DIS
LIN {X -0.109,Y -539.164,Z 546.188,A 0.000,B 0.000,C 90.000,E1 249.826} C_DIS
LIN {X -0.204,Y -536.260,Z 546.180,A 0.000,B 0.000,C 90.000,E1 248.411} C_DIS
LIN {X -0.143,Y -533.178,Z 546.172,A 0.000,B 0.000,C 90.000,E1 246.975} C_DIS
LIN {X 0.161,Y -530.550,Z 546.166,A 0.000,B 0.000,C 90.000,E1 245.793} C_DIS
LIN {X -0.066,Y -527.701,Z 546.159,A 0.000,B 0.000,C 90.000,E1 244.665} C_DIS
LIN {X -0.106,Y -524.757,Z 546.153,A 0.000,B 0.000,C 90.000,E1 243.512} C_DIS
LIN {X -0.188,Y -521.659,Z 546.146,A 0.000,B 0.000,C 90.000,E1 242.359} C_DIS
LIN {X -0.032,Y -516.875,Z 546.137,A 0.000,B 0.000,C 90.000,E1 240.589} C_DIS
LIN {X 0.011,Y -513.611,Z 546.130,A 0.000,B 0.000,C 90.000,E1 239.410} C_DIS
LIN {X 0.168,Y -509.165,Z 546.122,A 0.000,B 0.000,C 90.000,E1 237.916} C_DIS
LIN {X 0.246,Y -504.720,Z 546.114,A 0.000,B 0.000,C 90.000,E1 236.421} C_DIS
LIN {X -0.181,Y -500.344,Z 546.105,A 0.000,B 0.000,C 90.000,E1 234.975} C_DIS
LIN {X 0.022,Y -494.431,Z 546.094,A 0.000,B 0.000,C 90.000,E1 232.844} C_DIS
LIN {X 0.137,Y -491.133,Z 546.087,A 0.000,B 0.000,C 90.000,E1 231.618} C_DIS
LIN {X -0.060,Y -485.441,Z 546.075,A 0.000,B 0.000,C 90.000,E1 229.504} C_DIS
LIN {X 0.156,Y -480.674,Z 546.065,A 0.000,B 0.000,C 90.000,E1 227.634} C_DIS
LIN {X -0.021,Y -475.224,Z 546.053,A 0.000,B 0.000,C 90.000,E1 225.486} C_DIS
LIN {X -0.094,Y -470.724,Z 546.042,A 0.000,B 0.000,C 90.000,E1 223.623} C_DIS
LIN {X 0.163,Y -465.588,Z 546.030,A 0.000,B 0.000,C 90.000,E1 221.391} C_DIS
LIN {X 0.188,Y -461.965,Z 546.021,A 0.000,B 0.000,C 90.000,E1 219.806} C_DIS
LIN {X 0.110,Y -459.190,Z 546.014,A 0.000,B 0.000,C 90.000,E1 218.543} C_DIS
LIN {X -0.193,Y -454.993,Z 546.004,A 0.000,B 0.000,C 90.000,E1 216.664} C_DIS
LIN {X -0.145,Y -450.293,Z 545.991,A 0.000,B 0.000,C 90.000,E1 214.405} C_DIS
LIN {X 0.192,Y -446.368,Z 545.980,A 0.000,B 0.000,C 90.000,E1 212.418} C_DIS
LIN {X 0.080,Y -441.380,Z 545.966,A 0.000,B 0.000,C 90.000,E1 209.823} C_DIS
LIN {X 0.091,Y -438.420,Z 545.957,A 0.000,B 0.000,C 90.000,E1 208.180} C_DIS
LIN {X -0.143,Y -435.025,Z 545.946,A 0.000,B 0.000,C 90.000,E1 206.232} C_DIS
LIN {X -0.059,Y -431.198,Z 545.933,A 0.000,B 0.000,C 90.000,E1 203.898} C_DIS
LIN {X -0.060,Y -428.134,Z 545.922,A 0.000,B 0.000,C 90.000,E1 201.897} C_DIS
LIN {X 0.126,Y -423.947,Z 545.905,A 0.000,B 0.000,C 90.000,E1 198.852} C_DIS
LIN {X 0.073,Y -420.894,Z 545.892,A 0.000,B 0.000,C 90.000,E1 196.496} C_DIS
LIN {X 0.092,Y -418.086,Z 545.879,A 0.000,B 0.000,C 90.000,E1 194.120} C_DIS
LIN {X -0.003,Y -416.319,Z 545.871,A 0.000,B 0.000,C 90.000,E1 192.771} C_DIS
LIN {X 0.050,Y -413.705,Z 545.860,A 0.000,B 0.000,C 90.000,E1 190.715} C_DIS
LIN {X -0.118,Y -410.537,Z 545.844,A 0.000,B 0.000,C 90.000,E1 187.992} C_DIS
LIN {X -0.028,Y -407.738,Z 545.829,A 0.000,B 0.000,C 90.000,E1 185.220} C_DIS
LIN {X -0.113,Y -405.551,Z 545.816,A 0.000,B 0.000,C 90.000,E1 182.808} C_DIS
LIN {X 0.109,Y -403.624,Z 545.802,A 0.000,B 0.000,C 90.000,E1 180.344} C_DIS
LIN {X -0.120,Y -402.160,Z 545.789,A 0.000,B 0.000,C 90.000,E1 177.936} C_DIS
LIN {X 0.012,Y -401.015,Z 545.773,A 0.000,B 0.000,C 90.000,E1 175.122} C_DIS
LIN {X 0.174,Y -400.464,Z 545.757,A 0.000,B 0.000,C 90.000,E1 172.299} C_DIS
LIN {X 0.096,Y -400.333,Z 545.744,A 0.000,B 0.000,C 90.000,E1 169.859} C_DIS
LIN {X 0.102,Y -400.478,Z 545.732,A 0.000,B 0.000,C 90.000,E1 167.757} C_DIS
LIN {X -0.139,Y -401.062,Z 545.717,A 0.000,B 0.000,C 90.000,E1 164.991} C_DIS
LIN {X -0.230,Y -401.723,Z 545.705,A 0.000,B 0.000,C 90.000,E1 162.906} C_DIS
LIN {X 0.034,Y -402.766,Z 545.691,A 0.000,B 0.000,C 90.000,E1 160.423} C_DIS
LIN {X 0.128,Y -403.697,Z 545.682,A 0.000,B 0.000,C 90.000,E1 158.666} C_DIS
LIN {X 0.132,Y -405.059,Z 545.668,A 0.000,B 0.000,C 90.000,E1 156.230} C_DIS
LIN {X -0.180,Y -406.193,Z 545.658,A 0.000,B 0.000,C 90.000,E1 154.537} C_DIS
LIN {X 0.154,Y -407.545,Z 545.647,A 0.000,B 0.000,C 90.000,E1 152.410} C_DIS
LIN {X 0.161,Y -408.801,Z 545.635,A 0.000,B 0.000,C 90.000,E1 150.333} C_DIS
LIN {X -0.161,Y -409.516,Z 545.628,A 0.000,B 0.000,C 90.000,E1 148.997} C_DIS
LIN {X 0.017,Y -410.261,Z 545.618,A 0.000,B 0.000,C 90.000,E1 147.248} C_DIS
LIN {X 0.090,Y -410.894,Z 545.609,A 0.000,B 0.000,C 90.000,E1 145.515} C_DIS
LIN {X 0.010,Y -411.305,Z 545.601,A 0.000,B 0.000,C 90.000,E1 144.149} C_DIS
LIN {X -0.002,Y -411.660,Z 545.591,A 0.000,B 0.000,C 90.000,E1 142.431} C_DIS
LIN {X 0.080,Y -411.889,Z 545.584,A 0.000,B 0.000,C 90.000,E1 141.045} C_DIS
LIN {X 0.112,Y -411.990,Z 545.576,A 0.000,B 0.000,C 90.000,E1 139.666} C_DIS
LIN {X 0.045,Y -412.075,Z 545.567,A 0.000,B 0.000,C 90.000,E1 137.957} C_DIS
LIN {X 0.220,Y -412.130,Z 545.557,A 0.000,B 0.000,C 90.000,E1 136.215} C_DIS
LIN {X -0.033,Y -412.247,Z 545.546,A 0.000,B 0.000,C 90.000,E1 134.190} C_DIS
LIN {X 0.007,Y -412.374,Z 545.534,A 0.000,B 0.000,C 90.000,E1 132.123} C_DIS
LIN {X 0.049,Y -412.291,Z 545.526,A 0.000,B 0.000,C 90.000,E1 130.744} C_DIS
LIN {X -0.031,Y -412.106,Z 545.521,A 0.000,B 0.000,C 90.000,E1 129.725} C_DIS
LIN {X 0.063,Y -411.565,Z 545.513,A 0.000,B 0.000,C 90.000,E1 128.338} C_DIS
LIN {X 0.085,Y -411.109,Z 545.508,A 0.000,B 0.000,C 90.000,E1 127.443} C_DIS
LIN {X 0.045,Y -411.114,Z 545.508,A 0.000,B 0.000,C 90.000,E1 127.443} C_DIS
LIN {X 0.076,Y -415.617,Z 545.500,A 0.000,B 0.000,C 90.000,E1 125.931} C_DIS
LIN {X -0.065,Y -425.048,Z 545.479,A 0.000,B 0.000,C 90.000,E1 122.212} C_DIS
LIN {X -0.134,Y -431.000,Z 545.468,A 0.000,B 0.000,C 90.000,E1 120.207} C_DIS
LIN {X 0.012,Y -440.071,Z 545.448,A 0.000,B 0.000,C 90.000,E1 116.539} C_DIS
LIN {X 0.009,Y -444.853,Z 545.438,A 0.000,B 0.000,C 90.000,E1 114.899} C_DIS
LIN {X -0.106,Y -445.155,Z 545.438,A 0.000,B 0.000,C 90.000,E1 114.771} C_DIS
LIN {X -0.146,Y -445.182,Z 545.438,A 0.000,B 0.000,C 90.000,E1 114.771} C_DIS
LIN {X 0.126,Y -466.749,Z 545.432,A 0.000,B 0.000,C 90.000,E1 113.823} C_DIS
LIN {X -0.107,Y -484.163,Z 545.428,A 0.000,B 0.000,C 90.000,E1 113.131} C_DIS
LIN {X 0.248,Y -494.383,Z 545.426,A 0.000,B 0.000,C 90.000,E1 112.642} C_DIS
LIN {X 0.269,Y -501.136,Z 545.424,A 0.000,B 0.000,C 90.000,E1 112.333} C_DIS
LIN {X 0.162,Y -514.532,Z 545.421,A 0.000,B 0.000,C 90.000,E1 111.716} C_DIS
LIN {X 0.035,Y -521.220,Z 545.419,A 0.000,B 0.000,C 90.000,E1 111.408} C_DIS
LIN {X 0.237,Y -532.641,Z 545.416,A 0.000,B 0.000,C 90.000,E1 110.791} C_DIS
LIN {X -0.027,Y -540.676,Z 545.413,A 0.000,B 0.000,C 90.000,E1 110.375} C_DIS
LIN {X -0.004,Y -546.889,Z 545.411,A 0.000,B 0.000,C 90.000,E1 109.993} C_DIS
LIN {X 0.138,Y -552.897,Z 545.409,A 0.000,B 0.000,C 90.000,E1 109.577} C_DIS
LIN {X 0.064,Y -557.207,Z 545.407,A 0.000,B 0.000,C 90.000,E1 109.268} C_DIS
LIN {X -0.080,Y -564.019,Z 545.404,A 0.000,B 0.000,C 90.000,E1 108.725} C_DIS
LIN {X -0.063,Y -569.293,Z 545.401,A 0.000,B 0.000,C 90.000,E1 108.236} C_DIS
LIN {X 0.262,Y -574.323,Z 545.398,A 0.000,B 0.000,C 90.000,E1 107.692} C_DIS
LIN {X 0.205,Y -579.029,Z 545.396,A 0.000,B 0.000,C 90.000,E1 107.166} C_DIS
LIN {X -0.090,Y -585.281,Z 545.391,A 0.000,B 0.000,C 90.000,E1 106.386} C_DIS
LIN {X -0.097,Y -590.056,Z 545.387,A 0.000,B 0.000,C 90.000,E1 105.717} C_DIS
LIN {X -0.231,Y -594.490,Z 545.384,A 0.000,B 0.000,C 90.000,E1 105.064} C_DIS
LIN {X -0.255,Y -597.783,Z 545.381,A 0.000,B 0.000,C 90.000,E1 104.537} C_DIS
LIN {X 0.049,Y -602.349,Z 545.376,A 0.000,B 0.000,C 90.000,E1 103.716} C_DIS
LIN {X -0.245,Y -607.478,Z 545.371,A 0.000,B 0.000,C 90.000,E1 102.827} C_DIS
LIN {X -0.128,Y -611.030,Z 545.368,A 0.000,B 0.000,C 90.000,E1 102.175} C_DIS
LIN {X 0.066,Y -616.294,Z 545.362,A 0.000,B 0.000,C 90.000,E1 101.130} C_DIS
LIN {X 0.196,Y -618.696,Z 545.359,A 0.000,B 0.000,C 90.000,E1 100.602} C_DIS
LIN {X -0.158,Y -625.234,Z 545.351,A 0.000,B 0.000,C 90.000,E1 99.095} C_DIS
LIN {X -0.088,Y -630.638,Z 545.343,A 0.000,B 0.000,C 90.000,E1 97.814} C_DIS
LIN {X 0.179,Y -634.782,Z 545.338,A 0.000,B 0.000,C 90.000,E1 96.777} C_DIS
LIN {X -0.129,Y -638.854,Z 545.332,A 0.000,B 0.000,C 90.000,E1 95.796} C_DIS
LIN {X -0.198,Y -641.553,Z 545.328,A 0.000,B 0.000,C 90.000,E1 95.049} C_DIS
LIN {X 0.213,Y -644.767,Z 545.322,A 0.000,B 0.000,C 90.000,E1 94.012} C_DIS
LIN {X 0.163,Y -646.903,Z 545.318,A 0.000,B 0.000,C 90.000,E1 93.269} C_DIS
LIN {X 0.175,Y -648.834,Z 545.314,A 0.000,B 0.000,C 90.000,E1 92.522} C_DIS
LIN {X -0.259,Y -649.873,Z 545.311,A 0.000,B 0.000,C 90.000,E1 92.064} C_DIS
LIN {X -0.226,Y -651.177,Z 545.307,A 0.000,B 0.000,C 90.000,E1 91.318} C_DIS
LIN {X -0.199,Y -652.189,Z 545.303,A 0.000,B 0.000,C 90.000,E1 90.573} C_DIS
LIN {X -0.159,Y -652.847,Z 545.299,A 0.000,B 0.000,C 90.000,E1 89.828} C_DIS
LIN {X 0.291,Y -653.039,Z 545.298,A 0.000,B 0.000,C 90.000,E1 89.542} C_DIS
LIN {X 0.134,Y -653.155,Z 545.292,A 0.000,B 0.000,C 90.000,E1 88.568} C_DIS
LIN {X 0.200,Y -652.937,Z 545.288,A 0.000,B 0.000,C 90.000,E1 87.822} C_DIS
LIN {X -0.207,Y -652.644,Z 545.285,A 0.000,B 0.000,C 90.000,E1 87.364} C_DIS
LIN {X 0.303,Y -651.610,Z 545.280,A 0.000,B 0.000,C 90.000,E1 86.331} C_DIS
LIN {X -0.287,Y -650.555,Z 545.276,A 0.000,B 0.000,C 90.000,E1 85.641} C_DIS
LIN {X -0.238,Y -649.215,Z 545.272,A 0.000,B 0.000,C 90.000,E1 84.894} C_DIS
LIN {X 0.278,Y -647.210,Z 545.266,A 0.000,B 0.000,C 90.000,E1 83.856} C_DIS
LIN {X 0.287,Y -645.261,Z 545.262,A 0.000,B 0.000,C 90.000,E1 83.109} C_DIS
LIN {X -0.121,Y -643.849,Z 545.259,A 0.000,B 0.000,C 90.000,E1 82.648} C_DIS
LIN {X -0.234,Y -640.751,Z 545.254,A 0.000,B 0.000,C 90.000,E1 81.659} C_DIS
LIN {X -0.205,Y -638.132,Z 545.249,A 0.000,B 0.000,C 90.000,E1 80.905} C_DIS
LIN {X -0.203,Y -635.338,Z 545.245,A 0.000,B 0.000,C 90.000,E1 80.151} C_DIS
LIN {X 0.202,Y -631.254,Z 545.240,A 0.000,B 0.000,C 90.000,E1 79.106} C_DIS
LIN {X 0.248,Y -627.850,Z 545.235,A 0.000,B 0.000,C 90.000,E1 78.342} C_DIS
LIN {X 0.299,Y -624.916,Z 545.232,A 0.000,B 0.000,C 90.000,E1 77.701} C_DIS
LIN {X 0.281,Y -621.191,Z 545.228,A 0.000,B 0.000,C 90.000,E1 76.937} C_DIS
LIN {X -0.338,Y -617.820,Z 545.224,A 0.000,B 0.000,C 90.000,E1 76.353} C_DIS
LIN {X 0.118,Y -612.640,Z 545.219,A 0.000,B 0.000,C 90.000,E1 75.408} C_DIS
LIN {X 0.125,Y -607.703,Z 545.215,A 0.000,B 0.000,C 90.000,E1 74.629} C_DIS
LIN {X -0.080,Y -602.195,Z 545.210,A 0.000,B 0.000,C 90.000,E1 73.866} C_DIS
LIN {X 0.054,Y -597.125,Z 545.207,A 0.000,B 0.000,C 90.000,E1 73.196} C_DIS
LIN {X -0.028,Y -591.269,Z 545.203,A 0.000,B 0.000,C 90.000,E1 72.543} C_DIS
LIN {X 0.195,Y -587.629,Z 545.201,A 0.000,B 0.000,C 90.000,E1 72.127} C_DIS
LIN {X -0.116,Y -582.371,Z 545.198,A 0.000,B 0.000,C 90.000,E1 71.638} C_DIS
LIN {X 0.310,Y -576.824,Z 545.195,A 0.000,B 0.000,C 90.000,E1 71.094} C_DIS
LIN {X 0.316,Y -571.043,Z 545.192,A 0.000,B 0.000,C 90.000,E1 70.604} C_DIS
LIN {X 0.178,Y -565.510,Z 545.190,A 0.000,B 0.000,C 90.000,E1 70.188} C_DIS
LIN {X -0.086,Y -560.712,Z 545.188,A 0.000,B 0.000,C 90.000,E1 69.880} C_DIS
LIN {X -0.003,Y -555.918,Z 545.187,A 0.000,B 0.000,C 90.000,E1 69.571} C_DIS
LIN {X -0.011,Y -549.677,Z 545.185,A 0.000,B 0.000,C 90.000,E1 69.209} C_DIS
LIN {X 0.058,Y -542.958,Z 545.183,A 0.000,B 0.000,C 90.000,E1 68.847} C_DIS
LIN {X 0.063,Y -537.351,Z 545.181,A 0.000,B 0.000,C 90.000,E1 68.592} C_DIS
LIN {X 0.162,Y -532.029,Z 545.180,A 0.000,B 0.000,C 90.000,E1 68.358} C_DIS
LIN {X -0.017,Y -521.346,Z 545.178,A 0.000,B 0.000,C 90.000,E1 67.975} C_DIS
LIN {X -0.027,Y -512.496,Z 545.176,A 0.000,B 0.000,C 90.000,E1 67.667} C_DIS
LIN {X 0.114,Y -503.414,Z 545.174,A 0.000,B 0.000,C 90.000,E1 67.358} C_DIS
LIN {X 0.064,Y -487.280,Z 545.172,A 0.000,B 0.000,C 90.000,E1 66.869} C_DIS
LIN {X -0.130,Y -468.148,Z 545.168,A 0.000,B 0.000,C 90.000,E1 66.305} C_DIS
LIN {X 0.084,Y -463.543,Z 545.167,A 0.000,B 0.000,C 90.000,E1 66.125} C_DIS
LIN {X 0.242,Y -463.521,Z 545.167,A 0.000,B 0.000,C 90.000,E1 66.102} C_DIS
LIN {X 0.108,Y -455.497,Z 545.144,A 0.000,B 0.000,C 90.000,E1 61.897} C_DIS
LIN {X 0.114,Y -445.548,Z 545.119,A 0.000,B 0.000,C 90.000,E1 57.375} C_DIS
LIN {X -0.070,Y -443.757,Z 545.113,A 0.000,B 0.000,C 90.000,E1 56.421} C_DIS
LIN {X -0.027,Y -441.967,Z 545.110,A 0.000,B 0.000,C 90.000,E1 55.722} C_DIS
LIN {X -0.067,Y -441.961,Z 545.110,A 0.000,B 0.000,C 90.000,E1 55.722} C_DIS
LIN {X 0.057,Y -444.951,Z 545.101,A 0.000,B 0.000,C 90.000,E1 54.116} C_DIS
LIN {X -0.191,Y -447.259,Z 545.094,A 0.000,B 0.000,C 90.000,E1 52.844} C_DIS
LIN {X 0.201,Y -450.021,Z 545.084,A 0.000,B 0.000,C 90.000,E1 51.170} C_DIS
LIN {X -0.048,Y -452.578,Z 545.076,A 0.000,B 0.000,C 90.000,E1 49.585} C_DIS
LIN {X 0.089,Y -454.924,Z 545.067,A 0.000,B 0.000,C 90.000,E1 47.957} C_DIS
LIN {X 0.152,Y -456.211,Z 545.061,A 0.000,B 0.000,C 90.000,E1 46.986} C_DIS
LIN {X -0.079,Y -457.272,Z 545.056,A 0.000,B 0.000,C 90.000,E1 46.053} C_DIS
LIN {X 0.019,Y -458.155,Z 545.051,A 0.000,B 0.000,C 90.000,E1 45.081} C_DIS
LIN {X 0.165,Y -459.033,Z 545.043,A 0.000,B 0.000,C 90.000,E1 43.785} C_DIS
LIN {X -0.034,Y -459.550,Z 545.038,A 0.000,B 0.000,C 90.000,E1 42.852} C_DIS
LIN {X -0.226,Y -459.930,Z 545.033,A 0.000,B 0.000,C 90.000,E1 41.919} C_DIS
LIN {X -0.033,Y -460.168,Z 545.026,A 0.000,B 0.000,C 90.000,E1 40.620} C_DIS
LIN {X -0.133,Y -460.172,Z 545.019,A 0.000,B 0.000,C 90.000,E1 39.358} C_DIS
LIN {X -0.235,Y -460.034,Z 545.012,A 0.000,B 0.000,C 90.000,E1 38.096} C_DIS
LIN {X -0.132,Y -459.448,Z 545.001,A 0.000,B 0.000,C 90.000,E1 36.171} C_DIS
LIN {X -0.051,Y -458.682,Z 544.990,A 0.000,B 0.000,C 90.000,E1 34.246} C_DIS
LIN {X -0.131,Y -457.866,Z 544.980,A 0.000,B 0.000,C 90.000,E1 32.339} C_DIS
LIN {X 0.046,Y -457.203,Z 544.971,A 0.000,B 0.000,C 90.000,E1 30.718} C_DIS
LIN {X -0.136,Y -456.687,Z 544.964,A 0.000,B 0.000,C 90.000,E1 29.461} C_DIS
LIN {X -0.040,Y -455.985,Z 544.955,A 0.000,B 0.000,C 90.000,E1 27.847} C_DIS
LIN {X 0.049,Y -455.327,Z 544.946,A 0.000,B 0.000,C 90.000,E1 26.232} C_DIS
LIN {X 0.106,Y -454.265,Z 544.930,A 0.000,B 0.000,C 90.000,E1 23.334} C_DIS
LIN {X -0.023,Y -453.669,Z 544.917,A 0.000,B 0.000,C 90.000,E1 21.099} C_DIS
LIN {X -0.177,Y -453.156,Z 544.903,A 0.000,B 0.000,C 90.000,E1 18.544} C_DIS
LIN {X 0.123,Y -453.024,Z 544.887,A 0.000,B 0.000,C 90.000,E1 15.607} C_DIS
LIN {X 0.066,Y -453.322,Z 544.871,A 0.000,B 0.000,C 90.000,E1 12.715} C_DIS
LIN {X 0.043,Y -454.318,Z 544.853,A 0.000,B 0.000,C 90.000,E1 9.500} C_DIS
LIN {X 0.139,Y -455.340,Z 544.840,A 0.000,B 0.000,C 90.000,E1 7.239} C_DIS
LIN {X 0.044,Y -456.089,Z 544.833,A 0.000,B 0.000,C 90.000,E1 5.967} C_DIS
LIN {X -0.156,Y -457.367,Z 544.823,A 0.000,B 0.000,C 90.000,E1 4.069} C_DIS
LIN {X 0.022,Y -459.348,Z 544.808,A 0.000,B 0.000,C 90.000,E1 1.489} C_DIS
LIN {X 0.124,Y -461.693,Z 544.795,A 0.000,B 0.000,C 90.000,E1 359.141} C_DIS
LIN {X -0.205,Y -463.531,Z 544.787,A 0.000,B 0.000,C 90.000,E1 357.593} C_DIS
LIN {X 0.212,Y -466.017,Z 544.776,A 0.000,B 0.000,C 90.000,E1 355.641} C_DIS
LIN {X -0.208,Y -468.578,Z 544.765,A 0.000,B 0.000,C 90.000,E1 353.799} C_DIS
LIN {X 0.230,Y -471.491,Z 544.753,A 0.000,B 0.000,C 90.000,E1 351.546} C_DIS
LIN {X 0.181,Y -475.003,Z 544.739,A 0.000,B 0.000,C 90.000,E1 349.050} C_DIS
LIN {X 0.100,Y -478.505,Z 544.727,A 0.000,B 0.000,C 90.000,E1 346.881} C_DIS
LIN {X -0.099,Y -481.703,Z 544.717,A 0.000,B 0.000,C 90.000,E1 345.046} C_DIS
LIN {X -0.237,Y -485.641,Z 544.705,A 0.000,B 0.000,C 90.000,E1 342.906} C_DIS
LIN {X 0.132,Y -488.655,Z 544.696,A 0.000,B 0.000,C 90.000,E1 341.329} C_DIS
LIN {X -0.030,Y -492.248,Z 544.686,A 0.000,B 0.000,C 90.000,E1 339.518} C_DIS
LIN {X 0.227,Y -495.829,Z 544.676,A 0.000,B 0.000,C 90.000,E1 337.667} C_DIS
LIN {X 0.103,Y -499.303,Z 544.666,A 0.000,B 0.000,C 90.000,E1 335.869} C_DIS
LIN {X -0.272,Y -502.024,Z 544.658,A 0.000,B 0.000,C 90.000,E1 334.409} C_DIS
LIN {X 0.077,Y -504.729,Z 544.649,A 0.000,B 0.000,C 90.000,E1 332.871} C_DIS
LIN {X 0.029,Y -507.369,Z 544.641,A 0.000,B 0.000,C 90.000,E1 331.385} C_DIS
LIN {X -0.093,Y -510.516,Z 544.631,A 0.000,B 0.000,C 90.000,E1 329.616} C_DIS
LIN {X 0.031,Y -513.155,Z 544.623,A 0.000,B 0.000,C 90.000,E1 328.122} C_DIS
LIN {X -0.220,Y -516.887,Z 544.612,A 0.000,B 0.000,C 90.000,E1 326.087} C_DIS
LIN {X -0.169,Y -520.076,Z 544.602,A 0.000,B 0.000,C 90.000,E1 324.322} C_DIS
LIN {X -0.045,Y -523.223,Z 544.592,A 0.000,B 0.000,C 90.000,E1 322.557} C_DIS
LIN {X 0.011,Y -527.066,Z 544.581,A 0.000,B 0.000,C 90.000,E1 320.517} C_DIS
LIN {X 0.094,Y -531.173,Z 544.569,A 0.000,B 0.000,C 90.000,E1 318.485} C_DIS
LIN {X -0.166,Y -536.294,Z 544.557,A 0.000,B 0.000,C 90.000,E1 316.215} C_DIS
LIN {X 0.091,Y -542.467,Z 544.542,A 0.000,B 0.000,C 90.000,E1 313.623} C_DIS
LIN {X 0.113,Y -546.103,Z 544.535,A 0.000,B 0.000,C 90.000,E1 312.204} C_DIS
LIN {X 0.201,Y -548.801,Z 544.528,A 0.000,B 0.000,C 90.000,E1 311.067} C_DIS
LIN {X -0.078,Y -550.787,Z 544.524,A 0.000,B 0.000,C 90.000,E1 310.253} C_DIS
LIN {X 0.211,Y -554.910,Z 544.514,A 0.000,B 0.000,C 90.000,E1 308.543} C_DIS
LIN {X -0.139,Y -557.226,Z 544.510,A 0.000,B 0.000,C 90.000,E1 307.890} C_DIS
LIN {X 0.137,Y -560.495,Z 544.507,A 0.000,B 0.000,C 90.000,E1 307.282} C_DIS
LIN {X 0.142,Y -562.001,Z 544.506,A 0.000,B 0.000,C 90.000,E1 307.076} C_DIS
LIN {X 0.107,Y -565.291,Z 544.504,A 0.000,B 0.000,C 90.000,E1 306.710} C_DIS
LIN {X -0.234,Y -569.951,Z 544.502,A 0.000,B 0.000,C 90.000,E1 306.297} C_DIS
LIN {X -0.245,Y -576.367,Z 544.498,A 0.000,B 0.000,C 90.000,E1 305.724} C_DIS
LIN {X 0.142,Y -585.473,Z 544.494,A 0.000,B 0.000,C 90.000,E1 304.818} C_DIS
LIN {X -0.027,Y -590.462,Z 544.491,A 0.000,B 0.000,C 90.000,E1 304.326} C_DIS
LIN {X -0.118,Y -599.075,Z 544.486,A 0.000,B 0.000,C 90.000,E1 303.420} C_DIS
LIN {X -0.073,Y -607.455,Z 544.481,A 0.000,B 0.000,C 90.000,E1 302.498} C_DIS
LIN {X -0.142,Y -616.514,Z 544.475,A 0.000,B 0.000,C 90.000,E1 301.465} C_DIS
LIN {X 0.110,Y -623.067,Z 544.470,A 0.000,B 0.000,C 90.000,E1 300.669} C_DIS
LIN {X -0.116,Y -627.843,Z 544.467,A 0.000,B 0.000,C 90.000,E1 300.050} C_DIS
LIN {X -0.085,Y -631.261,Z 544.464,A 0.000,B 0.000,C 90.000,E1 299.539} C_DIS
LIN {X -0.006,Y -634.708,Z 544.461,A 0.000,B 0.000,C 90.000,E1 298.899} C_DIS
LIN {X -0.155,Y -637.532,Z 544.457,A 0.000,B 0.000,C 90.000,E1 298.281} C_DIS
LIN {X -0.055,Y -639.305,Z 544.454,A 0.000,B 0.000,C 90.000,E1 297.769} C_DIS
LIN {X 0.123,Y -641.692,Z 544.450,A 0.000,B 0.000,C 90.000,E1 297.001} C_DIS
LIN {X 0.256,Y -643.037,Z 544.447,A 0.000,B 0.000,C 90.000,E1 296.488} C_DIS
LIN {X 0.327,Y -643.557,Z 544.446,A 0.000,B 0.000,C 90.000,E1 296.232} C_DIS
LIN {X -0.106,Y -643.612,Z 544.443,A 0.000,B 0.000,C 90.000,E1 295.771} C_DIS
LIN {X -0.312,Y -643.457,Z 544.442,A 0.000,B 0.000,C 90.000,E1 295.540} C_DIS
LIN {X -0.162,Y -642.076,Z 544.439,A 0.000,B 0.000,C 90.000,E1 295.027} C_DIS
LIN {X -0.128,Y -641.529,Z 544.438,A 0.000,B 0.000,C 90.000,E1 294.899} C_DIS
LIN {X -0.059,Y -639.373,Z 544.437,A 0.000,B 0.000,C 90.000,E1 294.643} C_DIS
LIN {X -0.026,Y -638.241,Z 544.436,A 0.000,B 0.000,C 90.000,E1 294.515} C_DIS
LIN {X -0.093,Y -637.441,Z 544.435,A 0.000,B 0.000,C 90.000,E1 294.387} C_DIS
LIN {X -0.066,Y -636.103,Z 544.435,A 0.000,B 0.000,C 90.000,E1 294.259} C_DIS
LIN {X -0.040,Y -634.021,Z 544.434,A 0.000,B 0.000,C 90.000,E1 294.131} C_DIS
LIN {X 0.352,Y -632.071,Z 544.433,A 0.000,B 0.000,C 90.000,E1 293.951} C_DIS
LIN {X -0.091,Y -630.164,Z 544.432,A 0.000,B 0.000,C 90.000,E1 293.823} C_DIS
LIN {X 0.159,Y -623.009,Z 544.430,A 0.000,B 0.000,C 90.000,E1 293.387} C_DIS
LIN {X 0.134,Y -618.617,Z 544.429,A 0.000,B 0.000,C 90.000,E1 293.206} C_DIS
LIN {X -0.090,Y -610.308,Z 544.427,A 0.000,B 0.000,C 90.000,E1 292.898} C_DIS
LIN {X 0.077,Y -600.196,Z 544.425,A 0.000,B 0.000,C 90.000,E1 292.514} C_DIS
LIN {X 0.298,Y -583.096,Z 544.422,A 0.000,B 0.000,C 90.000,E1 291.897} C_DIS
LIN {X 0.199,Y -578.813,Z 544.421,A 0.000,B 0.000,C 90.000,E1 291.716} C_DIS
LIN {X 0.147,Y -576.353,Z 544.420,A 0.000,B 0.000,C 90.000,E1 291.589} C_DIS
LIN {X -0.006,Y -574.028,Z 544.419,A 0.000,B 0.000,C 90.000,E1 291.461} C_DIS
LIN {X -0.061,Y -571.829,Z 544.418,A 0.000,B 0.000,C 90.000,E1 291.280} C_DIS
LIN {X -0.116,Y -571.768,Z 544.418,A 0.000,B 0.000,C 90.000,E1 291.280} C_DIS
LIN {X -0.151,Y -570.988,Z 544.417,A 0.000,B 0.000,C 90.000,E1 291.025} C_DIS
LIN {X -0.091,Y -570.568,Z 544.414,A 0.000,B 0.000,C 90.000,E1 290.610} C_DIS
LIN {X 0.204,Y -570.617,Z 544.407,A 0.000,B 0.000,C 90.000,E1 289.214} C_DIS
LIN {X -0.045,Y -570.508,Z 544.399,A 0.000,B 0.000,C 90.000,E1 287.873} C_DIS
LIN {X 0.066,Y -570.200,Z 544.392,A 0.000,B 0.000,C 90.000,E1 286.496} C_DIS
LIN {X -0.162,Y -569.799,Z 544.386,A 0.000,B 0.000,C 90.000,E1 285.426} C_DIS
LIN {X 0.145,Y -568.720,Z 544.375,A 0.000,B 0.000,C 90.000,E1 283.480} C_DIS
LIN {X 0.262,Y -568.292,Z 544.370,A 0.000,B 0.000,C 90.000,E1 282.647} C_DIS
LIN {X 0.043,Y -567.585,Z 544.363,A 0.000,B 0.000,C 90.000,E1 281.299} C_DIS
LIN {X 0.088,Y -567.016,Z 544.357,A 0.000,B 0.000,C 90.000,E1 280.197} C_DIS
LIN {X 0.083,Y -566.033,Z 544.346,A 0.000,B 0.000,C 90.000,E1 278.276} C_DIS
LIN {X -0.114,Y -565.223,Z 544.335,A 0.000,B 0.000,C 90.000,E1 276.372} C_DIS
LIN {X -0.072,Y -564.713,Z 544.328,A 0.000,B 0.000,C 90.000,E1 274.992} C_DIS
LIN {X -0.141,Y -564.246,Z 544.322,A 0.000,B 0.000,C 90.000,E1 273.898} C_DIS
LIN {X -0.049,Y -563.390,Z 544.312,A 0.000,B 0.000,C 90.000,E1 272.236} C_DIS
LIN {X -0.075,Y -562.627,Z 544.305,A 0.000,B 0.000,C 90.000,E1 270.859} C_DIS
LIN {X -0.027,Y -561.593,Z 544.296,A 0.000,B 0.000,C 90.000,E1 269.198} C_DIS
LIN {X 0.009,Y -560.522,Z 544.286,A 0.000,B 0.000,C 90.000,E1 267.535} C_DIS
LIN {X -0.156,Y -559.811,Z 544.280,A 0.000,B 0.000,C 90.000,E1 266.445} C_DIS
LIN {X -0.001,Y -558.499,Z 544.269,A 0.000,B 0.000,C 90.000,E1 264.489} C_DIS
LIN {X 0.110,Y -557.079,Z 544.259,A 0.000,B 0.000,C 90.000,E1 262.534} C_DIS
LIN {X 0.007,Y -556.229,Z 544.252,A 0.000,B 0.000,C 90.000,E1 261.432} C_DIS
LIN {X -0.236,Y -555.342,Z 544.248,A 0.000,B 0.000,C 90.000,E1 260.622} C_DIS
LIN {X 0.238,Y -552.588,Z 544.235,A 0.000,B 0.000,C 90.000,E1 258.342} C_DIS
LIN {X 0.294,Y -550.892,Z 544.228,A 0.000,B 0.000,C 90.000,E1 256.937} C_DIS
LIN {X 0.014,Y -548.556,Z 544.218,A 0.000,B 0.000,C 90.000,E1 255.283} C_DIS
LIN {X 0.112,Y -546.536,Z 544.211,A 0.000,B 0.000,C 90.000,E1 253.866} C_DIS
LIN {X 0.236,Y -544.713,Z 544.204,A 0.000,B 0.000,C 90.000,E1 252.725} C_DIS
LIN {X 0.057,Y -542.214,Z 544.196,A 0.000,B 0.000,C 90.000,E1 251.329} C_DIS
LIN {X -0.160,Y -539.574,Z 544.188,A 0.000,B 0.000,C 90.000,E1 249.934} C_DIS
LIN {X 0.262,Y -536.677,Z 544.181,A 0.000,B 0.000,C 90.000,E1 248.465} C_DIS
LIN {X -0.163,Y -532.973,Z 544.171,A 0.000,B 0.000,C 90.000,E1 246.794} C_DIS
LIN {X 0.133,Y -530.270,Z 544.165,A 0.000,B 0.000,C 90.000,E1 245.613} C_DIS
LIN {X -0.277,Y -528.119,Z 544.160,A 0.000,B 0.000,C 90.000,E1 244.793} C_DIS
LIN {X 0.086,Y -524.403,Z 544.152,A 0.000,B 0.000,C 90.000,E1 243.307} C_DIS
LIN {X 0.001,Y -521.251,Z 544.145,A 0.000,B 0.000,C 90.000,E1 242.153} C_DIS
LIN {X 0.151,Y -516.458,Z 544.136,A 0.000,B 0.000,C 90.000,E1 240.383} C_DIS
LIN {X 0.188,Y -513.104,Z 544.129,A 0.000,B 0.000,C 90.000,E1 239.203} C_DIS
LIN {X 0.001,Y -509.568,Z 544.122,A 0.000,B 0.000,C 90.000,E1 238.043} C_DIS
LIN {X 0.090,Y -505.127,Z 544.114,A 0.000,B 0.000,C 90.000,E1 236.548} C_DIS
LIN {X 0.086,Y -500.777,Z 544.106,A 0.000,B 0.000,C 90.000,E1 235.055} C_DIS
LIN {X 0.153,Y -493.979,Z 544.093,A 0.000,B 0.000,C 90.000,E1 232.637} C_DIS
LIN {X -0.126,Y -490.629,Z 544.086,A 0.000,B 0.000,C 90.000,E1 231.457} C_DIS
LIN {X 0.041,Y -484.943,Z 544.074,A 0.000,B 0.000,C 90.000,E1 229.299} C_DIS
LIN {X -0.118,Y -480.186,Z 544.064,A 0.000,B 0.000,C 90.000,E1 227.472} C_DIS
LIN {X 0.036,Y -474.741,Z 544.052,A 0.000,B 0.000,C 90.000,E1 225.283} C_DIS
LIN {X -0.041,Y -470.231,Z 544.041,A 0.000,B 0.000,C 90.000,E1 223.419} C_DIS
LIN {X 0.106,Y -465.854,Z 544.031,A 0.000,B 0.000,C 90.000,E1 221.515} C_DIS
LIN {X 0.129,Y -462.227,Z 544.022,A 0.000,B 0.000,C 90.000,E1 219.930} C_DIS
LIN {X 0.050,Y -459.437,Z 544.015,A 0.000,B 0.000,C 90.000,E1 218.669} C_DIS
LIN {X 0.112,Y -454.522,Z 544.003,A 0.000,B 0.000,C 90.000,E1 216.423} C_DIS
LIN {X 0.082,Y -451.193,Z 543.994,A 0.000,B 0.000,C 90.000,E1 214.818} C_DIS
LIN {X 0.287,Y -448.527,Z 543.986,A 0.000,B 0.000,C 90.000,E1 213.499} C_DIS
LIN {X -0.041,Y -444.643,Z 543.976,A 0.000,B 0.000,C 90.000,E1 211.592} C_DIS
LIN {X 0.077,Y -440.999,Z 543.965,A 0.000,B 0.000,C 90.000,E1 209.617} C_DIS
LIN {X -0.063,Y -436.889,Z 543.952,A 0.000,B 0.000,C 90.000,E1 207.334} C_DIS
LIN {X 0.049,Y -433.567,Z 543.941,A 0.000,B 0.000,C 90.000,E1 205.335} C_DIS
LIN {X 0.099,Y -428.818,Z 543.924,A 0.000,B 0.000,C 90.000,E1 202.333} C_DIS
LIN {X -0.140,Y -424.913,Z 543.909,A 0.000,B 0.000,C 90.000,E1 199.685} C_DIS
LIN {X -0.133,Y -422.745,Z 543.900,A 0.000,B 0.000,C 90.000,E1 198.000} C_DIS
LIN {X 0.058,Y -419.793,Z 543.887,A 0.000,B 0.000,C 90.000,E1 195.607} C_DIS
LIN {X -0.158,Y -417.808,Z 543.877,A 0.000,B 0.000,C 90.000,E1 193.939} C_DIS
LIN {X -0.072,Y -415.156,Z 543.866,A 0.000,B 0.000,C 90.000,E1 191.883} C_DIS
LIN {X -0.129,Y -411.862,Z 543.851,A 0.000,B 0.000,C 90.000,E1 189.151} C_DIS
LIN {X 0.011,Y -409.593,Z 543.839,A 0.000,B 0.000,C 90.000,E1 187.068} C_DIS
LIN {X 0.054,Y -407.250,Z 543.826,A 0.000,B 0.000,C 90.000,E1 184.645} C_DIS
LIN {X -0.067,Y -405.166,Z 543.812,A 0.000,B 0.000,C 90.000,E1 182.236} C_DIS
LIN {X 0.009,Y -402.487,Z 543.791,A 0.000,B 0.000,C 90.000,E1 178.396} C_DIS
LIN {X 0.091,Y -401.160,Z 543.774,A 0.000,B 0.000,C 90.000,E1 175.241} C_DIS
LIN {X -0.102,Y -400.577,Z 543.758,A 0.000,B 0.000,C 90.000,E1 172.470} C_DIS
LIN {X 0.142,Y -400.453,Z 543.743,A 0.000,B 0.000,C 90.000,E1 169.634} C_DIS
LIN {X 0.227,Y -400.625,Z 543.731,A 0.000,B 0.000,C 90.000,E1 167.521} C_DIS
LIN {X -0.009,Y -401.258,Z 543.715,A 0.000,B 0.000,C 90.000,E1 164.755} C_DIS
LIN {X 0.083,Y -402.244,Z 543.700,A 0.000,B 0.000,C 90.000,E1 161.945} C_DIS
LIN {X 0.073,Y -403.601,Z 543.684,A 0.000,B 0.000,C 90.000,E1 159.156} C_DIS
LIN {X -0.150,Y -404.324,Z 543.677,A 0.000,B 0.000,C 90.000,E1 157.794} C_DIS
LIN {X 0.136,Y -406.070,Z 543.661,A 0.000,B 0.000,C 90.000,E1 154.973} C_DIS
LIN {X -0.077,Y -407.410,Z 543.650,A 0.000,B 0.000,C 90.000,E1 152.922} C_DIS
LIN {X 0.100,Y -408.290,Z 543.642,A 0.000,B 0.000,C 90.000,E1 151.513} C_DIS
LIN {X 0.044,Y -409.327,Z 543.632,A 0.000,B 0.000,C 90.000,E1 149.793} C_DIS
LIN {X 0.084,Y -409.977,Z 543.625,A 0.000,B 0.000,C 90.000,E1 148.408} C_DIS
LIN {X -0.080,Y -410.706,Z 543.615,A 0.000,B 0.000,C 90.000,E1 146.707} C_DIS
LIN {X -0.002,Y -411.315,Z 543.605,A 0.000,B 0.000,C 90.000,E1 144.975} C_DIS
LIN {X 0.241,Y -411.607,Z 543.600,A 0.000,B 0.000,C 90.000,E1 143.909} C_DIS
LIN {X 0.243,Y -411.974,Z 543.590,A 0.000,B 0.000,C 90.000,E1 142.190} C_DIS
LIN {X 0.015,Y -412.183,Z 543.583,A 0.000,B 0.000,C 90.000,E1 140.848} C_DIS
LIN {X 0.109,Y -412.291,Z 543.575,A 0.000,B 0.000,C 90.000,E1 139.461} C_DIS
LIN {X 0.013,Y -412.407,Z 543.565,A 0.000,B 0.000,C 90.000,E1 137.757} C_DIS
LIN {X 0.058,Y -412.470,Z 543.558,A 0.000,B 0.000,C 90.000,E1 136.377} C_DIS
LIN {X 0.257,Y -412.551,Z 543.544,A 0.000,B 0.000,C 90.000,E1 133.947} C_DIS
LIN {X 0.026,Y -412.681,Z 543.533,A 0.000,B 0.000,C 90.000,E1 131.919} C_DIS
LIN {X 0.077,Y -412.505,Z 543.525,A 0.000,B 0.000,C 90.000,E1 130.539} C_DIS
LIN {X 0.004,Y -412.254,Z 543.520,A 0.000,B 0.000,C 90.000,E1 129.519} C_DIS
LIN {X 0.191,Y -411.857,Z 543.514,A 0.000,B 0.000,C 90.000,E1 128.463} C_DIS
LIN {X 0.054,Y -411.257,Z 543.508,A 0.000,B 0.000,C 90.000,E1 127.397} C_DIS
LIN {X 0.015,Y -411.257,Z 543.508,A 0.000,B 0.000,C 90.000,E1 127.397} C_DIS
LIN {X -0.045,Y -415.182,Z 543.500,A 0.000,B 0.000,C 90.000,E1 126.091} C_DIS
LIN {X 0.065,Y -416.860,Z 543.497,A 0.000,B 0.000,C 90.000,E1 125.391} C_DIS
LIN {X -0.006,Y -426.576,Z 543.476,A 0.000,B 0.000,C 90.000,E1 121.671} C_DIS
LIN {X -0.043,Y -430.641,Z 543.469,A 0.000,B 0.000,C 90.000,E1 120.335} C_DIS
LIN {X -0.050,Y -441.544,Z 543.445,A 0.000,B 0.000,C 90.000,E1 116.027} C_DIS
LIN {X 0.077,Y -444.462,Z 543.439,A 0.000,B 0.000,C 90.000,E1 115.027} C_DIS
LIN {X 0.020,Y -445.758,Z 543.436,A 0.000,B 0.000,C 90.000,E1 114.463} C_DIS
LIN {X -0.019,Y -445.781,Z 543.436,A 0.000,B 0.000,C 90.000,E1 114.463} C_DIS
LIN {X -0.075,Y -470.392,Z 543.430,A 0.000,B 0.000,C 90.000,E1 113.439} C_DIS
LIN {X -0.141,Y -482.582,Z 543.427,A 0.000,B 0.000,C 90.000,E1 112.950} C_DIS
LIN {X -0.165,Y -492.813,Z 543.425,A 0.000,B 0.000,C 90.000,E1 112.514} C_DIS
LIN {X -0.081,Y -504.685,Z 543.422,A 0.000,B 0.000,C 90.000,E1 111.972} C_DIS
LIN {X 0.077,Y -514.839,Z 543.419,A 0.000,B 0.000,C 90.000,E1 111.482} C_DIS
LIN {X -0.103,Y -523.248,Z 543.417,A 0.000,B 0.000,C 90.000,E1 111.099} C_DIS
LIN {X -0.269,Y -533.087,Z 543.414,A 0.000,B 0.000,C 90.000,E1 110.610} C_DIS
LIN {X -0.119,Y -539.480,Z 543.412,A 0.000,B 0.000,C 90.000,E1 110.248} C_DIS
LIN {X -0.158,Y -545.712,Z 543.410,A 0.000,B 0.000,C 90.000,E1 109.885} C_DIS
LIN {X 0.275,Y -551.815,Z 543.408,A 0.000,B 0.000,C 90.000,E1 109.450} C_DIS
LIN {X -0.258,Y -557.658,Z 543.406,A 0.000,B 0.000,C 90.000,E1 109.087} C_DIS
LIN {X 0.128,Y -563.229,Z 543.403,A 0.000,B 0.000,C 90.000,E1 108.598} C_DIS
LIN {X 0.034,Y -568.577,Z 543.401,A 0.000,B 0.000,C 90.000,E1 108.127} C_DIS
LIN {X -0.106,Y -573.673,Z 543.398,A 0.000,B 0.000,C 90.000,E1 107.638} C_DIS
LIN {X 0.030,Y -578.493,Z 543.395,A 0.000,B 0.000,C 90.000,E1 107.094} C_DIS
LIN {X 0.058,Y -581.435,Z 543.393,A 0.000,B 0.000,C 90.000,E1 106.732} C_DIS
LIN {X -0.064,Y -585.560,Z 543.390,A 0.000,B 0.000,C 90.000,E1 106.205} C_DIS
LIN {X 0.009,Y -589.557,Z 543.387,A 0.000,B 0.000,C 90.000,E1 105.662} C_DIS
LIN {X -0.126,Y -594.125,Z 543.383,A 0.000,B 0.000,C 90.000,E1 105.009} C_DIS
LIN {X -0.223,Y -598.302,Z 543.380,A 0.000,B 0.000,C 90.000,E1 104.356} C_DIS
LIN {X 0.085,Y -602.992,Z 543.375,A 0.000,B 0.000,C 90.000,E1 103.536} C_DIS
LIN {X -0.001,Y -608.165,Z 543.370,A 0.000,B 0.000,C 90.000,E1 102.647} C_DIS
LIN {X -0.117,Y -611.827,Z 543.367,A 0.000,B 0.000,C 90.000,E1 102.007} C_DIS
LIN {X -0.259,Y -615.925,Z 543.362,A 0.000,B 0.000,C 90.000,E1 101.243} C_DIS
LIN {X 0.299,Y -619.039,Z 543.359,A 0.000,B 0.000,C 90.000,E1 100.546} C_DIS
LIN {X -0.115,Y -623.470,Z 543.353,A 0.000,B 0.000,C 90.000,E1 99.557} C_DIS
LIN {X 0.143,Y -627.918,Z 543.347,A 0.000,B 0.000,C 90.000,E1 98.511} C_DIS
LIN {X -0.253,Y -632.225,Z 543.342,A 0.000,B 0.000,C 90.000,E1 97.530} C_DIS
LIN {X -0.157,Y -637.410,Z 543.335,A 0.000,B 0.000,C 90.000,E1 96.258} C_DIS
LIN {X 0.016,Y -639.444,Z 543.332,A 0.000,B 0.000,C 90.000,E1 95.739} C_DIS
LIN {X -0.045,Y -642.188,Z 543.328,A 0.000,B 0.000,C 90.000,E1 94.992} C_DIS
LIN {X -0.267,Y -645.427,Z 543.322,A 0.000,B 0.000,C 90.000,E1 94.012} C_DIS
LIN {X -0.313,Y -647.601,Z 543.318,A 0.000,B 0.000,C 90.000,E1 93.269} C_DIS
LIN {X -0.295,Y -649.527,Z 543.314,A 0.000,B 0.000,C 90.000,E1 92.522} C_DIS
LIN {X -0.266,Y -651.041,Z 543.310,A 0.000,B 0.000,C 90.000,E1 91.776} C_DIS
LIN {X -0.243,Y -652.218,Z 543.306,A 0.000,B 0.000,C 90.000,E1 91.031} C_DIS
LIN {X -0.001,Y -652.851,Z 543.303,A 0.000,B 0.000,C 90.000,E1 90.516} C_DIS
LIN {X 0.046,Y -653.471,Z 543.299,A 0.000,B 0.000,C 90.000,E1 89.771} C_DIS
LIN {X 0.298,Y -653.707,Z 543.296,A 0.000,B 0.000,C 90.000,E1 89.255} C_DIS
LIN {X 0.148,Y -653.702,Z 543.291,A 0.000,B 0.000,C 90.000,E1 88.282} C_DIS
LIN {X 0.219,Y -653.323,Z 543.286,A 0.000,B 0.000,C 90.000,E1 87.535} C_DIS
LIN {X -0.188,Y -652.914,Z 543.284,A 0.000,B 0.000,C 90.000,E1 87.078} C_DIS
LIN {X -0.327,Y -651.741,Z 543.278,A 0.000,B 0.000,C 90.000,E1 86.102} C_DIS
LIN {X -0.269,Y -650.501,Z 543.274,A 0.000,B 0.000,C 90.000,E1 85.355} C_DIS
LIN {X -0.223,Y -649.084,Z 543.270,A 0.000,B 0.000,C 90.000,E1 84.609} C_DIS
LIN {X -0.126,Y -647.490,Z 543.266,A 0.000,B 0.000,C 90.000,E1 83.856} C_DIS
LIN {X -0.114,Y -645.490,Z 543.262,A 0.000,B 0.000,C 90.000,E1 83.109} C_DIS
LIN {X 0.119,Y -644.010,Z 543.259,A 0.000,B 0.000,C 90.000,E1 82.591} C_DIS
LIN {X 0.006,Y -640.876,Z 543.253,A 0.000,B 0.000,C 90.000,E1 81.602} C_DIS
LIN {X 0.034,Y -638.188,Z 543.249,A 0.000,B 0.000,C 90.000,E1 80.849} C_DIS
LIN {X -0.143,Y -634.267,Z 543.244,A 0.000,B 0.000,C 90.000,E1 79.859} C_DIS
LIN {X -0.185,Y -631.064,Z 543.239,A 0.000,B 0.000,C 90.000,E1 79.106} C_DIS
LIN {X -0.139,Y -627.568,Z 543.235,A 0.000,B 0.000,C 90.000,E1 78.342} C_DIS
LIN {X -0.089,Y -624.528,Z 543.232,A 0.000,B 0.000,C 90.000,E1 77.701} C_DIS
LIN {X -0.073,Y -621.356,Z 543.228,A 0.000,B 0.000,C 90.000,E1 77.061} C_DIS
LIN {X 0.053,Y -617.948,Z 543.225,A 0.000,B 0.000,C 90.000,E1 76.408} C_DIS
LIN {X -0.084,Y -612.605,Z 543.220,A 0.000,B 0.000,C 90.000,E1 75.519} C_DIS
LIN {X -0.232,Y -607.537,Z 543.215,A 0.000,B 0.000,C 90.000,E1 74.755} C_DIS
LIN {X 0.006,Y -602.107,Z 543.211,A 0.000,B 0.000,C 90.000,E1 73.976} C_DIS
LIN {X -0.162,Y -597.267,Z 543.208,A 0.000,B 0.000,C 90.000,E1 73.378} C_DIS
LIN {X -0.115,Y -591.438,Z 543.204,A 0.000,B 0.000,C 90.000,E1 72.725} C_DIS
LIN {X 0.045,Y -586.404,Z 543.201,A 0.000,B 0.000,C 90.000,E1 72.181} C_DIS
LIN {X -0.189,Y -581.054,Z 543.198,A 0.000,B 0.000,C 90.000,E1 71.692} C_DIS
LIN {X 0.168,Y -575.433,Z 543.195,A 0.000,B 0.000,C 90.000,E1 71.167} C_DIS
LIN {X -0.301,Y -571.178,Z 543.194,A 0.000,B 0.000,C 90.000,E1 70.859} C_DIS
LIN {X 0.059,Y -565.205,Z 543.191,A 0.000,B 0.000,C 90.000,E1 70.369} C_DIS
LIN {X 0.191,Y -558.824,Z 543.189,A 0.000,B 0.000,C 90.000,E1 69.934} C_DIS
LIN {X 0.131,Y -553.961,Z 543.187,A 0.000,B 0.000,C 90.000,E1 69.645} C_DIS
LIN {X 0.226,Y -547.146,Z 543.185,A 0.000,B 0.000,C 90.000,E1 69.263} C_DIS
LIN {X 0.024,Y -542.121,Z 543.184,A 0.000,B 0.000,C 90.000,E1 69.028} C_DIS
LIN {X 0.040,Y -534.940,Z 543.182,A 0.000,B 0.000,C 90.000,E1 68.720} C_DIS
LIN {X -0.157,Y -527.777,Z 543.180,A 0.000,B 0.000,C 90.000,E1 68.465} C_DIS
LIN {X 0.125,Y -516.970,Z 543.178,A 0.000,B 0.000,C 90.000,E1 68.050} C_DIS
LIN {X -0.129,Y -506.124,Z 543.176,A 0.000,B 0.000,C 90.000,E1 67.720} C_DIS
LIN {X 0.136,Y -496.897,Z 543.175,A 0.000,B 0.000,C 90.000,E1 67.411} C_DIS
LIN {X -0.153,Y -468.747,Z 543.170,A 0.000,B 0.000,C 90.000,E1 66.613} C_DIS
LIN {X 0.143,Y -464.340,Z 543.169,A 0.000,B 0.000,C 90.000,E1 66.433} C_DIS
LIN {X 0.114,Y -464.236,Z 543.169,A 0.000,B 0.000,C 90.000,E1 66.433} C_DIS
LIN {X 0.009,Y -456.012,Z 543.146,A 0.000,B 0.000,C 90.000,E1 62.231} C_DIS
LIN {X 0.114,Y -455.498,Z 543.144,A 0.000,B 0.000,C 90.000,E1 61.897} C_DIS
LIN {X 0.120,Y -445.549,Z 543.119,A 0.000,B 0.000,C 90.000,E1 57.375} C_DIS
LIN {X -0.064,Y -443.759,Z 543.113,A 0.000,B 0.000,C 90.000,E1 56.421} C_DIS
LIN {X -0.146,Y -442.331,Z 543.110,A 0.000,B 0.000,C 90.000,E1 55.881} C_DIS
LIN {X -0.186,Y -442.335,Z 543.110,A 0.000,B 0.000,C 90.000,E1 55.881} C_DIS
LIN {X 0.070,Y -445.686,Z 543.101,A 0.000,B 0.000,C 90.000,E1 54.116} C_DIS
LIN {X -0.165,Y -448.093,Z 543.094,A 0.000,B 0.000,C 90.000,E1 52.844} C_DIS
LIN {X 0.244,Y -450.892,Z 543.084,A 0.000,B 0.000,C 90.000,E1 51.170} C_DIS
LIN {X 0.068,Y -453.960,Z 543.074,A 0.000,B 0.000,C 90.000,E1 49.256} C_DIS
LIN {X -0.172,Y -455.817,Z 543.067,A 0.000,B 0.000,C 90.000,E1 48.000} C_DIS
LIN {X -0.072,Y -457.085,Z 543.061,A 0.000,B 0.000,C 90.000,E1 47.025} C_DIS
LIN {X -0.013,Y -457.844,Z 543.058,A 0.000,B 0.000,C 90.000,E1 46.377} C_DIS
LIN {X 0.090,Y -458.757,Z 543.052,A 0.000,B 0.000,C 90.000,E1 45.405} C_DIS
LIN {X 0.246,Y -459.668,Z 543.045,A 0.000,B 0.000,C 90.000,E1 44.109} C_DIS
LIN {X 0.054,Y -460.236,Z 543.040,A 0.000,B 0.000,C 90.000,E1 43.176} C_DIS
LIN {X -0.085,Y -460.712,Z 543.033,A 0.000,B 0.000,C 90.000,E1 41.919} C_DIS
LIN {X 0.121,Y -460.950,Z 543.026,A 0.000,B 0.000,C 90.000,E1 40.620} C_DIS
LIN {X 0.032,Y -460.949,Z 543.019,A 0.000,B 0.000,C 90.000,E1 39.358} C_DIS
LIN {X -0.058,Y -460.748,Z 543.012,A 0.000,B 0.000,C 90.000,E1 38.096} C_DIS
LIN {X 0.061,Y -460.131,Z 543.001,A 0.000,B 0.000,C 90.000,E1 36.171} C_DIS
LIN {X -0.217,Y -459.466,Z 542.992,A 0.000,B 0.000,C 90.000,E1 34.612} C_DIS
LIN {X -0.025,Y -458.649,Z 542.982,A 0.000,B 0.000,C 90.000,E1 32.673} C_DIS
LIN {X 0.167,Y -457.955,Z 542.973,A 0.000,B 0.000,C 90.000,E1 31.052} C_DIS
LIN {X -0.004,Y -457.438,Z 542.966,A 0.000,B 0.000,C 90.000,E1 29.795} C_DIS
LIN {X -0.187,Y -456.542,Z 542.955,A 0.000,B 0.000,C 90.000,E1 27.897} C_DIS
LIN {X -0.094,Y -455.833,Z 542.946,A 0.000,B 0.000,C 90.000,E1 26.283} C_DIS
LIN {X -0.009,Y -454.928,Z 542.934,A 0.000,B 0.000,C 90.000,E1 24.027} C_DIS
LIN {X 0.054,Y -454.258,Z 542.921,A 0.000,B 0.000,C 90.000,E1 21.770} C_DIS
LIN {X 0.021,Y -453.690,Z 542.909,A 0.000,B 0.000,C 90.000,E1 19.523} C_DIS
LIN {X -0.139,Y -453.347,Z 542.894,A 0.000,B 0.000,C 90.000,E1 16.968} C_DIS
LIN {X 0.078,Y -453.329,Z 542.883,A 0.000,B 0.000,C 90.000,E1 15.009} C_DIS
LIN {X 0.188,Y -453.526,Z 542.873,A 0.000,B 0.000,C 90.000,E1 13.063} C_DIS
LIN {X 0.186,Y -454.173,Z 542.858,A 0.000,B 0.000,C 90.000,E1 10.489} C_DIS
LIN {X 0.049,Y -455.227,Z 542.844,A 0.000,B 0.000,C 90.000,E1 7.936} C_DIS
LIN {X -0.109,Y -456.268,Z 542.833,A 0.000,B 0.000,C 90.000,E1 6.030} C_DIS
LIN {X -0.077,Y -457.703,Z 542.821,A 0.000,B 0.000,C 90.000,E1 3.784} C_DIS
LIN {X -0.078,Y -459.468,Z 542.809,A 0.000,B 0.000,C 90.000,E1 1.547} C_DIS
LIN {X 0.125,Y -461.818,Z 542.795,A 0.000,B 0.000,C 90.000,E1 359.141} C_DIS
LIN {X -0.201,Y -463.656,Z 542.787,A 0.000,B 0.000,C 90.000,E1 357.593} C_DIS
LIN {X 0.219,Y -466.133,Z 542.776,A 0.000,B 0.000,C 90.000,E1 355.641} C_DIS
LIN {X 0.073,Y -469.065,Z 542.764,A 0.000,B 0.000,C 90.000,E1 353.451} C_DIS
LIN {X 0.241,Y -471.559,Z 542.753,A 0.000,B 0.000,C 90.000,E1 351.546} C_DIS
LIN {X -0.108,Y -474.585,Z 542.741,A 0.000,B 0.000,C 90.000,E1 349.398} C_DIS
LIN {X -0.198,Y -478.018,Z 542.729,A 0.000,B 0.000,C 90.000,E1 347.229} C_DIS
LIN {X 0.062,Y -481.223,Z 542.719,A 0.000,B 0.000,C 90.000,E1 345.338} C_DIS
LIN {X -0.079,Y -485.146,Z 542.707,A 0.000,B 0.000,C 90.000,E1 343.196} C_DIS
LIN {X 0.151,Y -488.757,Z 542.696,A 0.000,B 0.000,C 90.000,E1 341.329} C_DIS
LIN {X -0.009,Y -492.350,Z 542.686,A 0.000,B 0.000,C 90.000,E1 339.518} C_DIS
LIN {X 0.250,Y -495.934,Z 542.676,A 0.000,B 0.000,C 90.000,E1 337.667} C_DIS
LIN {X 0.130,Y -499.428,Z 542.666,A 0.000,B 0.000,C 90.000,E1 335.869} C_DIS
LIN {X -0.244,Y -502.160,Z 542.658,A 0.000,B 0.000,C 90.000,E1 334.409} C_DIS
LIN {X 0.108,Y -504.890,Z 542.649,A 0.000,B 0.000,C 90.000,E1 332.871} C_DIS
LIN {X 0.062,Y -507.537,Z 542.641,A 0.000,B 0.000,C 90.000,E1 331.385} C_DIS
LIN {X -0.055,Y -510.697,Z 542.631,A 0.000,B 0.000,C 90.000,E1 329.616} C_DIS
LIN {X -0.287,Y -513.876,Z 542.621,A 0.000,B 0.000,C 90.000,E1 327.867} C_DIS
LIN {X -0.241,Y -517.631,Z 542.610,A 0.000,B 0.000,C 90.000,E1 325.801} C_DIS
LIN {X -0.116,Y -520.312,Z 542.602,A 0.000,B 0.000,C 90.000,E1 324.322} C_DIS
LIN {X 0.013,Y -523.489,Z 542.592,A 0.000,B 0.000,C 90.000,E1 322.557} C_DIS
LIN {X 0.077,Y -527.327,Z 542.581,A 0.000,B 0.000,C 90.000,E1 320.517} C_DIS
LIN {X -0.254,Y -532.020,Z 542.568,A 0.000,B 0.000,C 90.000,E1 318.243} C_DIS
LIN {X -0.086,Y -536.478,Z 542.557,A 0.000,B 0.000,C 90.000,E1 316.215} C_DIS
LIN {X 0.177,Y -542.578,Z 542.542,A 0.000,B 0.000,C 90.000,E1 313.623} C_DIS
LIN {X 0.201,Y -546.196,Z 542.535,A 0.000,B 0.000,C 90.000,E1 312.204} C_DIS
LIN {X 0.291,Y -548.924,Z 542.528,A 0.000,B 0.000,C 90.000,E1 311.067} C_DIS
LIN {X 0.015,Y -550.838,Z 542.524,A 0.000,B 0.000,C 90.000,E1 310.253} C_DIS
LIN {X -0.060,Y -555.551,Z 542.513,A 0.000,B 0.000,C 90.000,E1 308.302} C_DIS
LIN {X -0.018,Y -557.384,Z 542.509,A 0.000,B 0.000,C 90.000,E1 307.684} C_DIS
LIN {X 0.066,Y -558.838,Z 542.508,A 0.000,B 0.000,C 90.000,E1 307.397} C_DIS
LIN {X -0.293,Y -559.887,Z 542.506,A 0.000,B 0.000,C 90.000,E1 307.156} C_DIS
LIN {X 0.013,Y -562.680,Z 542.504,A 0.000,B 0.000,C 90.000,E1 306.710} C_DIS
LIN {X 0.112,Y -565.071,Z 542.502,A 0.000,B 0.000,C 90.000,E1 306.423} C_DIS
LIN {X 0.236,Y -570.252,Z 542.500,A 0.000,B 0.000,C 90.000,E1 305.884} C_DIS
LIN {X 0.056,Y -576.924,Z 542.496,A 0.000,B 0.000,C 90.000,E1 305.264} C_DIS
LIN {X 0.328,Y -583.298,Z 542.492,A 0.000,B 0.000,C 90.000,E1 304.612} C_DIS
LIN {X 0.089,Y -589.591,Z 542.489,A 0.000,B 0.000,C 90.000,E1 303.992} C_DIS
LIN {X 0.007,Y -596.949,Z 542.485,A 0.000,B 0.000,C 90.000,E1 303.214} C_DIS
LIN {X 0.324,Y -606.492,Z 542.479,A 0.000,B 0.000,C 90.000,E1 302.133} C_DIS
LIN {X -0.092,Y -615.526,Z 542.473,A 0.000,B 0.000,C 90.000,E1 301.131} C_DIS
LIN {X 0.157,Y -620.953,Z 542.469,A 0.000,B 0.000,C 90.000,E1 300.463} C_DIS
LIN {X -0.398,Y -625.762,Z 542.466,A 0.000,B 0.000,C 90.000,E1 299.873} C_DIS
LIN {X -0.070,Y -629.156,Z 542.463,A 0.000,B 0.000,C 90.000,E1 299.333} C_DIS
LIN {X -0.012,Y -632.604,Z 542.459,A 0.000,B 0.000,C 90.000,E1 298.693} C_DIS
LIN {X 0.100,Y -635.912,Z 542.455,A 0.000,B 0.000,C 90.000,E1 297.924} C_DIS
LIN {X -0.027,Y -638.298,Z 542.451,A 0.000,B 0.000,C 90.000,E1 297.180} C_DIS
LIN {X 0.138,Y -640.263,Z 542.447,A 0.000,B 0.000,C 90.000,E1 296.411} C_DIS
LIN {X -0.020,Y -640.409,Z 542.444,A 0.000,B 0.000,C 90.000,E1 295.924} C_DIS
LIN {X 0.044,Y -640.316,Z 542.443,A 0.000,B 0.000,C 90.000,E1 295.668} C_DIS
LIN {X 0.107,Y -639.689,Z 542.441,A 0.000,B 0.000,C 90.000,E1 295.412} C_DIS
LIN {X 0.170,Y -639.258,Z 542.440,A 0.000,B 0.000,C 90.000,E1 295.155} C_DIS
LIN {X 0.201,Y -638.889,Z 542.439,A 0.000,B 0.000,C 90.000,E1 295.027} C_DIS
LIN {X 0.258,Y -637.036,Z 542.438,A 0.000,B 0.000,C 90.000,E1 294.771} C_DIS
LIN {X 0.311,Y -635.734,Z 542.436,A 0.000,B 0.000,C 90.000,E1 294.515} C_DIS
LIN {X 0.336,Y -634.791,Z 542.436,A 0.000,B 0.000,C 90.000,E1 294.387} C_DIS
LIN {X 0.120,Y -631.831,Z 542.434,A 0.000,B 0.000,C 90.000,E1 294.155} C_DIS
LIN {X 0.199,Y -629.777,Z 542.433,A 0.000,B 0.000,C 90.000,E1 293.951} C_DIS
LIN {X 0.270,Y -628.077,Z 542.433,A 0.000,B 0.000,C 90.000,E1 293.823} C_DIS
LIN {X -0.167,Y -621.366,Z 542.430,A 0.000,B 0.000,C 90.000,E1 293.462} C_DIS
LIN {X 0.190,Y -617.518,Z 542.429,A 0.000,B 0.000,C 90.000,E1 293.259} C_DIS
LIN {X -0.080,Y -615.532,Z 542.429,A 0.000,B 0.000,C 90.000,E1 293.206} C_DIS
LIN {X -0.131,Y -612.779,Z 542.428,A 0.000,B 0.000,C 90.000,E1 293.078} C_DIS
LIN {X 0.159,Y -609.130,Z 542.427,A 0.000,B 0.000,C 90.000,E1 292.898} C_DIS
LIN {X 0.241,Y -599.250,Z 542.425,A 0.000,B 0.000,C 90.000,E1 292.514} C_DIS
LIN {X -0.033,Y -585.976,Z 542.423,A 0.000,B 0.000,C 90.000,E1 292.078} C_DIS
LIN {X -0.178,Y -580.001,Z 542.421,A 0.000,B 0.000,C 90.000,E1 291.844} C_DIS
LIN {X -0.311,Y -574.413,Z 542.419,A 0.000,B 0.000,C 90.000,E1 291.535} C_DIS
LIN {X 0.309,Y -572.233,Z 542.418,A 0.000,B 0.000,C 90.000,E1 291.280} C_DIS
LIN {X 0.271,Y -572.201,Z 542.418,A 0.000,B 0.000,C 90.000,E1 291.280} C_DIS
LIN {X 0.146,Y -571.739,Z 542.418,A 0.000,B 0.000,C 90.000,E1 291.153} C_DIS
LIN {X -0.111,Y -571.390,Z 542.417,A 0.000,B 0.000,C 90.000,E1 290.972} C_DIS
LIN {X 0.237,Y -571.107,Z 542.414,A 0.000,B 0.000,C 90.000,E1 290.429} C_DIS
LIN {X -0.350,Y -571.211,Z 542.408,A 0.000,B 0.000,C 90.000,E1 289.396} C_DIS
LIN {X -0.044,Y -571.161,Z 542.400,A 0.000,B 0.000,C 90.000,E1 288.000} C_DIS
LIN {X 0.083,Y -570.873,Z 542.392,A 0.000,B 0.000,C 90.000,E1 286.622} C_DIS
LIN {X 0.234,Y -570.611,Z 542.388,A 0.000,B 0.000,C 90.000,E1 285.788} C_DIS
LIN {X -0.030,Y -569.774,Z 542.379,A 0.000,B 0.000,C 90.000,E1 284.175} C_DIS
LIN {X -0.041,Y -568.896,Z 542.370,A 0.000,B 0.000,C 90.000,E1 282.535} C_DIS
LIN {X -0.242,Y -568.222,Z 542.362,A 0.000,B 0.000,C 90.000,E1 281.186} C_DIS
LIN {X -0.084,Y -567.636,Z 542.356,A 0.000,B 0.000,C 90.000,E1 280.074} C_DIS
LIN {X -0.167,Y -566.649,Z 542.345,A 0.000,B 0.000,C 90.000,E1 278.163} C_DIS
LIN {X 0.121,Y -565.956,Z 542.336,A 0.000,B 0.000,C 90.000,E1 276.486} C_DIS
LIN {X 0.172,Y -565.488,Z 542.328,A 0.000,B 0.000,C 90.000,E1 275.106} C_DIS
LIN {X 0.218,Y -564.899,Z 542.321,A 0.000,B 0.000,C 90.000,E1 273.726} C_DIS
LIN {X 0.218,Y -564.157,Z 542.313,A 0.000,B 0.000,C 90.000,E1 272.350} C_DIS
LIN {X 0.205,Y -563.405,Z 542.306,A 0.000,B 0.000,C 90.000,E1 270.974} C_DIS
LIN {X 0.166,Y -562.498,Z 542.298,A 0.000,B 0.000,C 90.000,E1 269.599} C_DIS
LIN {X 0.223,Y -561.407,Z 542.289,A 0.000,B 0.000,C 90.000,E1 267.936} C_DIS
LIN {X 0.255,Y -560.302,Z 542.279,A 0.000,B 0.000,C 90.000,E1 266.274} C_DIS
LIN {X -0.270,Y -559.175,Z 542.270,A 0.000,B 0.000,C 90.000,E1 264.666} C_DIS
LIN {X -0.147,Y -557.890,Z 542.261,A 0.000,B 0.000,C 90.000,E1 262.989} C_DIS
LIN {X -0.173,Y -556.830,Z 542.253,A 0.000,B 0.000,C 90.000,E1 261.602} C_DIS
LIN {X 0.143,Y -555.984,Z 542.249,A 0.000,B 0.000,C 90.000,E1 260.735} C_DIS
LIN {X -0.137,Y -553.569,Z 542.238,A 0.000,B 0.000,C 90.000,E1 258.814} C_DIS
LIN {X 0.053,Y -551.520,Z 542.229,A 0.000,B 0.000,C 90.000,E1 257.117} C_DIS
LIN {X 0.208,Y -549.615,Z 542.221,A 0.000,B 0.000,C 90.000,E1 255.700} C_DIS
LIN {X -0.202,Y -547.580,Z 542.213,A 0.000,B 0.000,C 90.000,E1 254.338} C_DIS
LIN {X -0.058,Y -545.780,Z 542.207,A 0.000,B 0.000,C 90.000,E1 253.196} C_DIS
LIN {X 0.064,Y -543.828,Z 542.200,A 0.000,B 0.000,C 90.000,E1 252.054} C_DIS
LIN {X -0.124,Y -541.222,Z 542.193,A 0.000,B 0.000,C 90.000,E1 250.659} C_DIS
LIN {X -0.080,Y -538.995,Z 542.186,A 0.000,B 0.000,C 90.000,E1 249.518} C_DIS
LIN {X -0.176,Y -536.038,Z 542.178,A 0.000,B 0.000,C 90.000,E1 248.103} C_DIS
LIN {X -0.119,Y -532.890,Z 542.170,A 0.000,B 0.000,C 90.000,E1 246.666} C_DIS
LIN {X 0.177,Y -530.141,Z 542.164,A 0.000,B 0.000,C 90.000,E1 245.485} C_DIS
LIN {X 0.169,Y -527.232,Z 542.158,A 0.000,B 0.000,C 90.000,E1 244.332} C_DIS
LIN {X -0.110,Y -524.198,Z 542.151,A 0.000,B 0.000,C 90.000,E1 243.204} C_DIS
LIN {X 0.037,Y -521.022,Z 542.145,A 0.000,B 0.000,C 90.000,E1 242.025} C_DIS
LIN {X 0.182,Y -516.206,Z 542.135,A 0.000,B 0.000,C 90.000,E1 240.255} C_DIS
LIN {X 0.213,Y -512.823,Z 542.128,A 0.000,B 0.000,C 90.000,E1 239.076} C_DIS
LIN {X 0.019,Y -509.296,Z 542.122,A 0.000,B 0.000,C 90.000,E1 237.916} C_DIS
LIN {X 0.100,Y -504.856,Z 542.114,A 0.000,B 0.000,C 90.000,E1 236.421} C_DIS
LIN {X -0.323,Y -500.497,Z 542.105,A 0.000,B 0.000,C 90.000,E1 234.975} C_DIS
LIN {X -0.254,Y -493.693,Z 542.092,A 0.000,B 0.000,C 90.000,E1 232.557} C_DIS
LIN {X 0.002,Y -491.182,Z 542.087,A 0.000,B 0.000,C 90.000,E1 231.618} C_DIS
LIN {X 0.177,Y -485.469,Z 542.075,A 0.000,B 0.000,C 90.000,E1 229.461} C_DIS
LIN {X 0.027,Y -480.672,Z 542.065,A 0.000,B 0.000,C 90.000,E1 227.634} C_DIS
LIN {X -0.149,Y -475.216,Z 542.053,A 0.000,B 0.000,C 90.000,E1 225.486} C_DIS
LIN {X -0.221,Y -470.678,Z 542.042,A 0.000,B 0.000,C 90.000,E1 223.623} C_DIS
LIN {X 0.279,Y -466.284,Z 542.032,A 0.000,B 0.000,C 90.000,E1 221.676} C_DIS
LIN {X 0.061,Y -461.933,Z 542.021,A 0.000,B 0.000,C 90.000,E1 219.806} C_DIS
LIN {X -0.017,Y -459.107,Z 542.014,A 0.000,B 0.000,C 90.000,E1 218.543} C_DIS
LIN {X 0.045,Y -454.253,Z 542.002,A 0.000,B 0.000,C 90.000,E1 216.297} C_DIS
LIN {X -0.272,Y -450.261,Z 541.991,A 0.000,B 0.000,C 90.000,E1 214.405} C_DIS
LIN {X 0.134,Y -445.650,Z 541.978,A 0.000,B 0.000,C 90.000,E1 212.084} C_DIS
LIN {X 0.121,Y -441.965,Z 541.968,A 0.000,B 0.000,C 90.000,E1 210.129} C_DIS
LIN {X 0.031,Y -437.221,Z 541.953,A 0.000,B 0.000,C 90.000,E1 207.513} C_DIS
LIN {X -0.035,Y -433.328,Z 541.940,A 0.000,B 0.000,C 90.000,E1 205.207} C_DIS
LIN {X 0.005,Y -428.600,Z 541.923,A 0.000,B 0.000,C 90.000,E1 202.206} C_DIS
LIN {X 0.013,Y -424.703,Z 541.909,A 0.000,B 0.000,C 90.000,E1 199.523} C_DIS
LIN {X 0.157,Y -422.552,Z 541.899,A 0.000,B 0.000,C 90.000,E1 197.819} C_DIS
LIN {X -0.009,Y -419.216,Z 541.884,A 0.000,B 0.000,C 90.000,E1 195.134} C_DIS
LIN {X 0.016,Y -417.601,Z 541.877,A 0.000,B 0.000,C 90.000,E1 193.772} C_DIS
LIN {X 0.107,Y -415.002,Z 541.865,A 0.000,B 0.000,C 90.000,E1 191.715} C_DIS
LIN {X 0.083,Y -412.134,Z 541.852,A 0.000,B 0.000,C 90.000,E1 189.321} C_DIS
LIN {X -0.185,Y -409.857,Z 541.840,A 0.000,B 0.000,C 90.000,E1 187.296} C_DIS
LIN {X -0.174,Y -407.481,Z 541.827,A 0.000,B 0.000,C 90.000,E1 184.878} C_DIS
LIN {X 0.146,Y -405.380,Z 541.814,A 0.000,B 0.000,C 90.000,E1 182.407} C_DIS
LIN {X -0.138,Y -402.871,Z 541.794,A 0.000,B 0.000,C 90.000,E1 178.969} C_DIS
LIN {X -0.080,Y -401.322,Z 541.775,A 0.000,B 0.000,C 90.000,E1 175.469} C_DIS
LIN {X 0.086,Y -400.707,Z 541.759,A 0.000,B 0.000,C 90.000,E1 172.648} C_DIS
LIN {X -0.010,Y -400.588,Z 541.742,A 0.000,B 0.000,C 90.000,E1 169.511} C_DIS
LIN {X -0.016,Y -400.822,Z 541.728,A 0.000,B 0.000,C 90.000,E1 167.061} C_DIS
LIN {X -0.157,Y -401.522,Z 541.713,A 0.000,B 0.000,C 90.000,E1 164.283} C_DIS
LIN {X -0.030,Y -402.427,Z 541.699,A 0.000,B 0.000,C 90.000,E1 161.819} C_DIS
LIN {X -0.124,Y -403.644,Z 541.685,A 0.000,B 0.000,C 90.000,E1 159.390} C_DIS
LIN {X 0.128,Y -404.577,Z 541.676,A 0.000,B 0.000,C 90.000,E1 157.614} C_DIS
LIN {X 0.051,Y -406.338,Z 541.660,A 0.000,B 0.000,C 90.000,E1 154.845} C_DIS
LIN {X 0.207,Y -407.704,Z 541.649,A 0.000,B 0.000,C 90.000,E1 152.743} C_DIS
LIN {X -0.058,Y -408.818,Z 541.639,A 0.000,B 0.000,C 90.000,E1 151.051} C_DIS
LIN {X -0.026,Y -409.630,Z 541.632,A 0.000,B 0.000,C 90.000,E1 149.665} C_DIS
LIN {X 0.016,Y -410.284,Z 541.624,A 0.000,B 0.000,C 90.000,E1 148.280} C_DIS
LIN {X 0.082,Y -411.035,Z 541.614,A 0.000,B 0.000,C 90.000,E1 146.548} C_DIS
LIN {X -0.064,Y -411.621,Z 541.605,A 0.000,B 0.000,C 90.000,E1 144.848} C_DIS
LIN {X 0.013,Y -412.001,Z 541.597,A 0.000,B 0.000,C 90.000,E1 143.463} C_DIS
LIN {X 0.028,Y -412.345,Z 541.588,A 0.000,B 0.000,C 90.000,E1 141.743} C_DIS
LIN {X -0.021,Y -412.595,Z 541.578,A 0.000,B 0.000,C 90.000,E1 140.033} C_DIS
LIN {X 0.072,Y -412.701,Z 541.570,A 0.000,B 0.000,C 90.000,E1 138.647} C_DIS
LIN {X -0.161,Y -412.820,Z 541.559,A 0.000,B 0.000,C 90.000,E1 136.620} C_DIS
LIN {X 0.046,Y -412.910,Z 541.546,A 0.000,B 0.000,C 90.000,E1 134.190} C_DIS
LIN {X 0.102,Y -412.978,Z 541.534,A 0.000,B 0.000,C 90.000,E1 132.123} C_DIS
LIN {X -0.116,Y -412.830,Z 541.527,A 0.000,B 0.000,C 90.000,E1 130.782} C_DIS
LIN {X 0.080,Y -412.582,Z 541.521,A 0.000,B 0.000,C 90.000,E1 129.725} C_DIS
LIN {X -0.141,Y -411.991,Z 541.513,A 0.000,B 0.000,C 90.000,E1 128.382} C_DIS
LIN {X -0.141,Y -411.426,Z 541.508,A 0.000,B 0.000,C 90.000,E1 127.363} C_DIS
LIN {X -0.180,Y -411.435,Z 541.508,A 0.000,B 0.000,C 90.000,E1 127.363} C_DIS
LIN {X 0.160,Y -415.891,Z 541.499,A 0.000,B 0.000,C 90.000,E1 125.804} C_DIS
LIN {X 0.043,Y -425.368,Z 541.478,A 0.000,B 0.000,C 90.000,E1 122.084} C_DIS
LIN {X -0.013,Y -430.384,Z 541.469,A 0.000,B 0.000,C 90.000,E1 120.413} C_DIS
LIN {X -0.009,Y -431.992,Z 541.465,A 0.000,B 0.000,C 90.000,E1 119.745} C_DIS
LIN {X -0.017,Y -441.312,Z 541.445,A 0.000,B 0.000,C 90.000,E1 116.104} C_DIS
LIN {X 0.111,Y -444.215,Z 541.440,A 0.000,B 0.000,C 90.000,E1 115.103} C_DIS
LIN {X 0.153,Y -445.087,Z 541.438,A 0.000,B 0.000,C 90.000,E1 114.771} C_DIS
LIN {X 0.112,Y -446.386,Z 541.434,A 0.000,B 0.000,C 90.000,E1 114.155} C_DIS
LIN {X 0.072,Y -446.488,Z 541.434,A 0.000,B 0.000,C 90.000,E1 114.155} C_DIS
LIN {X 0.130,Y -478.648,Z 541.427,A 0.000,B 0.000,C 90.000,E1 112.823} C_DIS
LIN {X 0.037,Y -488.986,Z 541.425,A 0.000,B 0.000,C 90.000,E1 112.408} C_DIS
LIN {X -0.017,Y -499.223,Z 541.422,A 0.000,B 0.000,C 90.000,E1 111.972} C_DIS
LIN {X 0.245,Y -511.083,Z 541.419,A 0.000,B 0.000,C 90.000,E1 111.408} C_DIS
LIN {X 0.128,Y -522.946,Z 541.416,A 0.000,B 0.000,C 90.000,E1 110.865} C_DIS
LIN {X -0.037,Y -534.436,Z 541.413,A 0.000,B 0.000,C 90.000,E1 110.301} C_DIS
LIN {X -0.287,Y -539.295,Z 541.411,A 0.000,B 0.000,C 90.000,E1 110.066} C_DIS
LIN {X -0.096,Y -545.546,Z 541.409,A 0.000,B 0.000,C 90.000,E1 109.685} C_DIS
LIN {X 0.192,Y -551.633,Z 541.407,A 0.000,B 0.000,C 90.000,E1 109.268} C_DIS
LIN {X 0.176,Y -557.581,Z 541.405,A 0.000,B 0.000,C 90.000,E1 108.852} C_DIS
LIN {X 0.026,Y -563.263,Z 541.402,A 0.000,B 0.000,C 90.000,E1 108.417} C_DIS
LIN {X -0.061,Y -568.684,Z 541.400,A 0.000,B 0.000,C 90.000,E1 107.946} C_DIS
LIN {X -0.223,Y -572.658,Z 541.398,A 0.000,B 0.000,C 90.000,E1 107.583} C_DIS
LIN {X 0.321,Y -578.501,Z 541.394,A 0.000,B 0.000,C 90.000,E1 106.913} C_DIS
LIN {X -0.281,Y -582.873,Z 541.391,A 0.000,B 0.000,C 90.000,E1 106.441} C_DIS
LIN {X -0.093,Y -588.828,Z 541.387,A 0.000,B 0.000,C 90.000,E1 105.662} C_DIS
LIN {X -0.234,Y -593.538,Z 541.383,A 0.000,B 0.000,C 90.000,E1 105.009} C_DIS
LIN {X -0.051,Y -599.497,Z 541.378,A 0.000,B 0.000,C 90.000,E1 104.064} C_DIS
LIN {X 0.209,Y -605.048,Z 541.373,A 0.000,B 0.000,C 90.000,E1 103.119} C_DIS
LIN {X 0.003,Y -609.626,Z 541.369,A 0.000,B 0.000,C 90.000,E1 102.355} C_DIS
LIN {X -0.099,Y -613.253,Z 541.365,A 0.000,B 0.000,C 90.000,E1 101.715} C_DIS
LIN {X 0.012,Y -616.057,Z 541.362,A 0.000,B 0.000,C 90.000,E1 101.186} C_DIS
LIN {X -0.093,Y -619.849,Z 541.358,A 0.000,B 0.000,C 90.000,E1 100.423} C_DIS
LIN {X 0.110,Y -624.356,Z 541.352,A 0.000,B 0.000,C 90.000,E1 99.378} C_DIS
LIN {X -0.339,Y -628.878,Z 541.347,A 0.000,B 0.000,C 90.000,E1 98.398} C_DIS
LIN {X -0.297,Y -634.245,Z 541.339,A 0.000,B 0.000,C 90.000,E1 97.125} C_DIS
LIN {X -0.171,Y -639.502,Z 541.332,A 0.000,B 0.000,C 90.000,E1 95.853} C_DIS
LIN {X 0.160,Y -643.188,Z 541.327,A 0.000,B 0.000,C 90.000,E1 94.821} C_DIS
LIN {X -0.048,Y -646.416,Z 541.321,A 0.000,B 0.000,C 90.000,E1 93.841} C_DIS
LIN {X -0.044,Y -648.599,Z 541.317,A 0.000,B 0.000,C 90.000,E1 93.094} C_DIS
LIN {X -0.051,Y -650.478,Z 541.313,A 0.000,B 0.000,C 90.000,E1 92.350} C_DIS
LIN {X -0.012,Y -651.908,Z 541.309,A 0.000,B 0.000,C 90.000,E1 91.604} C_DIS
LIN {X 0.021,Y -653.055,Z 541.305,A 0.000,B 0.000,C 90.000,E1 90.859} C_DIS
LIN {X 0.069,Y -653.876,Z 541.301,A 0.000,B 0.000,C 90.000,E1 90.115} C_DIS
LIN {X 0.126,Y -654.282,Z 541.297,A 0.000,B 0.000,C 90.000,E1 89.370} C_DIS
LIN {X 0.184,Y -654.338,Z 541.292,A 0.000,B 0.000,C 90.000,E1 88.625} C_DIS
LIN {X 0.262,Y -654.163,Z 541.288,A 0.000,B 0.000,C 90.000,E1 87.879} C_DIS
LIN {X 0.313,Y -653.577,Z 541.284,A 0.000,B 0.000,C 90.000,E1 87.135} C_DIS
LIN {X -0.263,Y -652.676,Z 541.280,A 0.000,B 0.000,C 90.000,E1 86.445} C_DIS
LIN {X -0.192,Y -651.651,Z 541.276,A 0.000,B 0.000,C 90.000,E1 85.698} C_DIS
LIN {X 0.297,Y -649.679,Z 541.271,A 0.000,B 0.000,C 90.000,E1 84.666} C_DIS
LIN {X -0.246,Y -648.093,Z 541.266,A 0.000,B 0.000,C 90.000,E1 83.970} C_DIS
LIN {X 0.257,Y -645.362,Z 541.261,A 0.000,B 0.000,C 90.000,E1 82.932} C_DIS
LIN {X -0.147,Y -643.769,Z 541.258,A 0.000,B 0.000,C 90.000,E1 82.470} C_DIS
LIN {X 0.286,Y -640.469,Z 541.253,A 0.000,B 0.000,C 90.000,E1 81.432} C_DIS
LIN {X -0.152,Y -638.683,Z 541.250,A 0.000,B 0.000,C 90.000,E1 80.971} C_DIS
LIN {X -0.331,Y -634.714,Z 541.244,A 0.000,B 0.000,C 90.000,E1 79.982} C_DIS
LIN {X 0.179,Y -630.266,Z 541.239,A 0.000,B 0.000,C 90.000,E1 78.926} C_DIS
LIN {X -0.109,Y -625.485,Z 541.233,A 0.000,B 0.000,C 90.000,E1 77.937} C_DIS
LIN {X -0.122,Y -621.603,Z 541.229,A 0.000,B 0.000,C 90.000,E1 77.173} C_DIS
LIN {X 0.009,Y -618.153,Z 541.225,A 0.000,B 0.000,C 90.000,E1 76.520} C_DIS
LIN {X -0.273,Y -612.665,Z 541.220,A 0.000,B 0.000,C 90.000,E1 75.644} C_DIS
LIN {X -0.325,Y -606.686,Z 541.215,A 0.000,B 0.000,C 90.000,E1 74.755} C_DIS
LIN {X -0.085,Y -602.009,Z 541.212,A 0.000,B 0.000,C 90.000,E1 74.102} C_DIS
LIN {X 0.107,Y -597.686,Z 541.209,A 0.000,B 0.000,C 90.000,E1 73.559} C_DIS
LIN {X -0.180,Y -595.453,Z 541.207,A 0.000,B 0.000,C 90.000,E1 73.323} C_DIS
LIN {X 0.030,Y -591.828,Z 541.205,A 0.000,B 0.000,C 90.000,E1 72.906} C_DIS
LIN {X -0.148,Y -585.776,Z 541.202,A 0.000,B 0.000,C 90.000,E1 72.308} C_DIS
LIN {X 0.084,Y -580.764,Z 541.199,A 0.000,B 0.000,C 90.000,E1 71.819} C_DIS
LIN {X 0.164,Y -573.798,Z 541.196,A 0.000,B 0.000,C 90.000,E1 71.221} C_DIS
LIN {X 0.153,Y -570.882,Z 541.195,A 0.000,B 0.000,C 90.000,E1 70.986} C_DIS
LIN {X 0.145,Y -565.017,Z 541.192,A 0.000,B 0.000,C 90.000,E1 70.550} C_DIS
LIN {X -0.265,Y -558.845,Z 541.190,A 0.000,B 0.000,C 90.000,E1 70.188} C_DIS
LIN {X -0.090,Y -552.606,Z 541.188,A 0.000,B 0.000,C 90.000,E1 69.806} C_DIS
LIN {X 0.065,Y -547.540,Z 541.186,A 0.000,B 0.000,C 90.000,E1 69.518} C_DIS
LIN {X 0.063,Y -542.435,Z 541.185,A 0.000,B 0.000,C 90.000,E1 69.263} C_DIS
LIN {X 0.095,Y -535.201,Z 541.183,A 0.000,B 0.000,C 90.000,E1 68.954} C_DIS
LIN {X -0.266,Y -528.019,Z 541.182,A 0.000,B 0.000,C 90.000,E1 68.720} C_DIS
LIN {X -0.187,Y -517.212,Z 541.180,A 0.000,B 0.000,C 90.000,E1 68.337} C_DIS
LIN {X -0.038,Y -508.076,Z 541.178,A 0.000,B 0.000,C 90.000,E1 68.028} C_DIS
LIN {X 0.076,Y -498.921,Z 541.176,A 0.000,B 0.000,C 90.000,E1 67.741} C_DIS
LIN {X -0.071,Y -482.784,Z 541.174,A 0.000,B 0.000,C 90.000,E1 67.305} C_DIS
LIN {X -0.149,Y -465.064,Z 541.171,A 0.000,B 0.000,C 90.000,E1 66.794} C_DIS
LIN {X -0.176,Y -464.990,Z 541.171,A 0.000,B 0.000,C 90.000,E1 66.794} C_DIS
LIN {X 0.005,Y -456.516,Z 541.147,A 0.000,B 0.000,C 90.000,E1 62.538} C_DIS
LIN {X 0.006,Y -455.473,Z 541.144,A 0.000,B 0.000,C 90.000,E1 61.897} C_DIS
LIN {X 0.013,Y -445.524,Z 541.119,A 0.000,B 0.000,C 90.000,E1 57.375} C_DIS
LIN {X -0.171,Y -443.722,Z 541.113,A 0.000,B 0.000,C 90.000,E1 56.421} C_DIS
LIN {X -0.053,Y -442.687,Z 541.111,A 0.000,B 0.000,C 90.000,E1 56.008} C_DIS
LIN {X -0.092,Y -442.692,Z 541.111,A 0.000,B 0.000,C 90.000,E1 56.008} C_DIS
LIN {X 0.284,Y -445.838,Z 541.102,A 0.000,B 0.000,C 90.000,E1 54.402} C_DIS
LIN {X -0.248,Y -448.949,Z 541.093,A 0.000,B 0.000,C 90.000,E1 52.844} C_DIS
LIN {X -0.166,Y -451.217,Z 541.086,A 0.000,B 0.000,C 90.000,E1 51.537} C_DIS
LIN {X -0.114,Y -452.788,Z 541.081,A 0.000,B 0.000,C 90.000,E1 50.561} C_DIS
LIN {X 0.022,Y -454.878,Z 541.074,A 0.000,B 0.000,C 90.000,E1 49.256} C_DIS
LIN {X -0.206,Y -456.730,Z 541.067,A 0.000,B 0.000,C 90.000,E1 48.000} C_DIS
LIN {X -0.063,Y -458.371,Z 541.059,A 0.000,B 0.000,C 90.000,E1 46.701} C_DIS
LIN {X 0.084,Y -459.603,Z 541.052,A 0.000,B 0.000,C 90.000,E1 45.405} C_DIS
LIN {X 0.255,Y -460.509,Z 541.045,A 0.000,B 0.000,C 90.000,E1 44.109} C_DIS
LIN {X 0.072,Y -461.047,Z 541.040,A 0.000,B 0.000,C 90.000,E1 43.176} C_DIS
LIN {X -0.055,Y -461.497,Z 541.033,A 0.000,B 0.000,C 90.000,E1 41.919} C_DIS
LIN {X 0.163,Y -461.732,Z 541.026,A 0.000,B 0.000,C 90.000,E1 40.620} C_DIS
LIN {X 0.086,Y -461.705,Z 541.019,A 0.000,B 0.000,C 90.000,E1 39.358} C_DIS
LIN {X 0.007,Y -461.456,Z 541.012,A 0.000,B 0.000,C 90.000,E1 38.096} C_DIS
LIN {X 0.027,Y -460.920,Z 541.003,A 0.000,B 0.000,C 90.000,E1 36.503} C_DIS
LIN {X 0.275,Y -460.557,Z 540.998,A 0.000,B 0.000,C 90.000,E1 35.518} C_DIS
LIN {X 0.112,Y -459.701,Z 540.987,A 0.000,B 0.000,C 90.000,E1 33.627} C_DIS
LIN {X -0.064,Y -459.002,Z 540.978,A 0.000,B 0.000,C 90.000,E1 32.054} C_DIS
LIN {X 0.012,Y -458.160,Z 540.967,A 0.000,B 0.000,C 90.000,E1 30.129} C_DIS
LIN {X -0.153,Y -457.245,Z 540.957,A 0.000,B 0.000,C 90.000,E1 28.231} C_DIS
LIN {X -0.040,Y -456.495,Z 540.948,A 0.000,B 0.000,C 90.000,E1 26.616} C_DIS
LIN {X -0.157,Y -455.528,Z 540.935,A 0.000,B 0.000,C 90.000,E1 24.387} C_DIS
LIN {X 0.066,Y -454.673,Z 540.921,A 0.000,B 0.000,C 90.000,E1 21.791} C_DIS
LIN {X -0.216,Y -454.079,Z 540.909,A 0.000,B 0.000,C 90.000,E1 19.577} C_DIS
LIN {X -0.068,Y -453.687,Z 540.894,A 0.000,B 0.000,C 90.000,E1 16.985} C_DIS
LIN {X 0.048,Y -453.631,Z 540.882,A 0.000,B 0.000,C 90.000,E1 14.717} C_DIS
LIN {X -0.037,Y -453.782,Z 540.873,A 0.000,B 0.000,C 90.000,E1 13.119} C_DIS
LIN {X -0.035,Y -454.408,Z 540.859,A 0.000,B 0.000,C 90.000,E1 10.546} C_DIS
LIN {X -0.169,Y -455.433,Z 540.844,A 0.000,B 0.000,C 90.000,E1 7.992} C_DIS
LIN {X 0.128,Y -456.438,Z 540.834,A 0.000,B 0.000,C 90.000,E1 6.030} C_DIS
LIN {X 0.165,Y -457.839,Z 540.821,A 0.000,B 0.000,C 90.000,E1 3.784} C_DIS
LIN {X 0.169,Y -459.599,Z 540.809,A 0.000,B 0.000,C 90.000,E1 1.547} C_DIS
LIN {X 0.125,Y -461.943,Z 540.795,A 0.000,B 0.000,C 90.000,E1 359.141} C_DIS
LIN {X -0.197,Y -463.781,Z 540.787,A 0.000,B 0.000,C 90.000,E1 357.593} C_DIS
LIN {X -0.023,Y -466.640,Z 540.774,A 0.000,B 0.000,C 90.000,E1 355.355} C_DIS
LIN {X 0.082,Y -469.146,Z 540.764,A 0.000,B 0.000,C 90.000,E1 353.451} C_DIS
LIN {X 0.075,Y -472.065,Z 540.752,A 0.000,B 0.000,C 90.000,E1 351.254} C_DIS
LIN {X 0.206,Y -475.136,Z 540.739,A 0.000,B 0.000,C 90.000,E1 349.050} C_DIS
LIN {X -0.024,Y -479.137,Z 540.726,A 0.000,B 0.000,C 90.000,E1 346.589} C_DIS
LIN {X 0.236,Y -482.963,Z 540.714,A 0.000,B 0.000,C 90.000,E1 344.393} C_DIS
LIN {X -0.200,Y -485.817,Z 540.705,A 0.000,B 0.000,C 90.000,E1 342.906} C_DIS
LIN {X 0.172,Y -488.859,Z 540.696,A 0.000,B 0.000,C 90.000,E1 341.329} C_DIS
LIN {X 0.014,Y -492.462,Z 540.686,A 0.000,B 0.000,C 90.000,E1 339.518} C_DIS
LIN {X -0.182,Y -496.058,Z 540.676,A 0.000,B 0.000,C 90.000,E1 337.720} C_DIS
LIN {X -0.234,Y -500.114,Z 540.664,A 0.000,B 0.000,C 90.000,E1 335.613} C_DIS
LIN {X 0.077,Y -502.831,Z 540.656,A 0.000,B 0.000,C 90.000,E1 334.076} C_DIS
LIN {X -0.231,Y -505.588,Z 540.648,A 0.000,B 0.000,C 90.000,E1 332.615} C_DIS
LIN {X -0.022,Y -508.223,Z 540.639,A 0.000,B 0.000,C 90.000,E1 331.101} C_DIS
LIN {X -0.115,Y -511.418,Z 540.630,A 0.000,B 0.000,C 90.000,E1 329.331} C_DIS
LIN {X 0.110,Y -514.618,Z 540.620,A 0.000,B 0.000,C 90.000,E1 327.533} C_DIS
LIN {X -0.188,Y -517.875,Z 540.610,A 0.000,B 0.000,C 90.000,E1 325.801} C_DIS
LIN {X -0.058,Y -520.556,Z 540.602,A 0.000,B 0.000,C 90.000,E1 324.322} C_DIS
LIN {X 0.036,Y -524.289,Z 540.590,A 0.000,B 0.000,C 90.000,E1 322.271} C_DIS
LIN {X 0.149,Y -527.593,Z 540.581,A 0.000,B 0.000,C 90.000,E1 320.517} C_DIS
LIN {X 0.160,Y -532.888,Z 540.566,A 0.000,B 0.000,C 90.000,E1 317.919} C_DIS
LIN {X 0.358,Y -537.319,Z 540.555,A 0.000,B 0.000,C 90.000,E1 315.891} C_DIS
LIN {X 0.270,Y -542.690,Z 540.543,A 0.000,B 0.000,C 90.000,E1 313.623} C_DIS
LIN {X -0.069,Y -546.282,Z 540.535,A 0.000,B 0.000,C 90.000,E1 312.243} C_DIS
LIN {X 0.029,Y -549.031,Z 540.528,A 0.000,B 0.000,C 90.000,E1 311.105} C_DIS
LIN {X 0.113,Y -550.942,Z 540.524,A 0.000,B 0.000,C 90.000,E1 310.253} C_DIS
LIN {X 0.338,Y -554.058,Z 540.516,A 0.000,B 0.000,C 90.000,E1 308.830} C_DIS
LIN {X 0.058,Y -557.160,Z 540.509,A 0.000,B 0.000,C 90.000,E1 307.604} C_DIS
LIN {X 0.076,Y -559.237,Z 540.506,A 0.000,B 0.000,C 90.000,E1 306.996} C_DIS
LIN {X -0.041,Y -560.709,Z 540.504,A 0.000,B 0.000,C 90.000,E1 306.790} C_DIS
LIN {X 0.052,Y -562.271,Z 540.503,A 0.000,B 0.000,C 90.000,E1 306.503} C_DIS
LIN {X 0.170,Y -564.631,Z 540.501,A 0.000,B 0.000,C 90.000,E1 306.217} C_DIS
LIN {X -0.037,Y -566.540,Z 540.500,A 0.000,B 0.000,C 90.000,E1 305.964} C_DIS
LIN {X -0.250,Y -572.087,Z 540.497,A 0.000,B 0.000,C 90.000,E1 305.391} C_DIS
LIN {X -0.379,Y -582.042,Z 540.491,A 0.000,B 0.000,C 90.000,E1 304.405} C_DIS
LIN {X 0.165,Y -588.321,Z 540.487,A 0.000,B 0.000,C 90.000,E1 303.706} C_DIS
LIN {X -0.290,Y -595.649,Z 540.483,A 0.000,B 0.000,C 90.000,E1 302.959} C_DIS
LIN {X 0.028,Y -605.152,Z 540.477,A 0.000,B 0.000,C 90.000,E1 301.878} C_DIS
LIN {X -0.385,Y -613.041,Z 540.472,A 0.000,B 0.000,C 90.000,E1 301.003} C_DIS
LIN {X -0.130,Y -617.407,Z 540.469,A 0.000,B 0.000,C 90.000,E1 300.463} C_DIS
LIN {X -0.162,Y -620.507,Z 540.467,A 0.000,B 0.000,C 90.000,E1 300.079} C_DIS
LIN {X 0.130,Y -625.000,Z 540.464,A 0.000,B 0.000,C 90.000,E1 299.411} C_DIS
LIN {X 0.143,Y -627.566,Z 540.461,A 0.000,B 0.000,C 90.000,E1 299.027} C_DIS
LIN {X -0.060,Y -630.858,Z 540.458,A 0.000,B 0.000,C 90.000,E1 298.409} C_DIS
LIN {X -0.034,Y -632.001,Z 540.456,A 0.000,B 0.000,C 90.000,E1 298.153} C_DIS
LIN {X 0.029,Y -633.947,Z 540.454,A 0.000,B 0.000,C 90.000,E1 297.641} C_DIS
LIN {X 0.066,Y -634.789,Z 540.452,A 0.000,B 0.000,C 90.000,E1 297.385} C_DIS
LIN {X 0.199,Y -636.695,Z 540.448,A 0.000,B 0.000,C 90.000,E1 296.616} C_DIS
LIN {X 0.298,Y -637.103,Z 540.445,A 0.000,B 0.000,C 90.000,E1 296.104} C_DIS
LIN {X 0.350,Y -637.221,Z 540.444,A 0.000,B 0.000,C 90.000,E1 295.848} C_DIS
LIN {X -0.123,Y -636.506,Z 540.441,A 0.000,B 0.000,C 90.000,E1 295.387} C_DIS
LIN {X -0.344,Y -635.802,Z 540.440,A 0.000,B 0.000,C 90.000,E1 295.155} C_DIS
LIN {X -0.247,Y -633.420,Z 540.437,A 0.000,B 0.000,C 90.000,E1 294.643} C_DIS
LIN {X -0.226,Y -632.472,Z 540.436,A 0.000,B 0.000,C 90.000,E1 294.515} C_DIS
LIN {X -0.160,Y -628.612,Z 540.434,A 0.000,B 0.000,C 90.000,E1 294.131} C_DIS
LIN {X -0.079,Y -627.273,Z 540.433,A 0.000,B 0.000,C 90.000,E1 294.003} C_DIS
LIN {X -0.124,Y -622.316,Z 540.432,A 0.000,B 0.000,C 90.000,E1 293.695} C_DIS
LIN {X -0.085,Y -621.149,Z 540.431,A 0.000,B 0.000,C 90.000,E1 293.590} C_DIS
LIN {X 0.161,Y -616.773,Z 540.430,A 0.000,B 0.000,C 90.000,E1 293.334} C_DIS
LIN {X 0.075,Y -614.720,Z 540.429,A 0.000,B 0.000,C 90.000,E1 293.259} C_DIS
LIN {X 0.163,Y -611.407,Z 540.428,A 0.000,B 0.000,C 90.000,E1 293.078} C_DIS
LIN {X -0.293,Y -603.124,Z 540.426,A 0.000,B 0.000,C 90.000,E1 292.770} C_DIS
LIN {X 0.084,Y -595.848,Z 540.425,A 0.000,B 0.000,C 90.000,E1 292.461} C_DIS
LIN {X 0.267,Y -589.002,Z 540.424,A 0.000,B 0.000,C 90.000,E1 292.206} C_DIS
LIN {X 0.089,Y -579.781,Z 540.421,A 0.000,B 0.000,C 90.000,E1 291.844} C_DIS
LIN {X -0.063,Y -574.423,Z 540.420,A 0.000,B 0.000,C 90.000,E1 291.535} C_DIS
LIN {X -0.250,Y -572.764,Z 540.419,A 0.000,B 0.000,C 90.000,E1 291.408} C_DIS
LIN {X 0.157,Y -571.966,Z 540.417,A 0.000,B 0.000,C 90.000,E1 291.046} C_DIS
LIN {X 0.339,Y -571.677,Z 540.414,A 0.000,B 0.000,C 90.000,E1 290.482} C_DIS
LIN {X -0.243,Y -571.794,Z 540.408,A 0.000,B 0.000,C 90.000,E1 289.450} C_DIS
LIN {X 0.070,Y -571.783,Z 540.400,A 0.000,B 0.000,C 90.000,E1 288.055} C_DIS
LIN {X 0.204,Y -571.524,Z 540.393,A 0.000,B 0.000,C 90.000,E1 286.677} C_DIS
LIN {X -0.006,Y -571.160,Z 540.387,A 0.000,B 0.000,C 90.000,E1 285.607} C_DIS
LIN {X -0.035,Y -570.483,Z 540.379,A 0.000,B 0.000,C 90.000,E1 284.245} C_DIS
LIN {X -0.265,Y -569.509,Z 540.369,A 0.000,B 0.000,C 90.000,E1 282.355} C_DIS
LIN {X -0.100,Y -568.589,Z 540.358,A 0.000,B 0.000,C 90.000,E1 280.423} C_DIS
LIN {X 0.105,Y -567.240,Z 540.344,A 0.000,B 0.000,C 90.000,E1 277.936} C_DIS
LIN {X 0.217,Y -566.364,Z 540.330,A 0.000,B 0.000,C 90.000,E1 275.454} C_DIS
LIN {X -0.131,Y -565.646,Z 540.321,A 0.000,B 0.000,C 90.000,E1 273.841} C_DIS
LIN {X -0.228,Y -565.059,Z 540.315,A 0.000,B 0.000,C 90.000,E1 272.751} C_DIS
LIN {X -0.119,Y -564.147,Z 540.306,A 0.000,B 0.000,C 90.000,E1 271.088} C_DIS
LIN {X 0.206,Y -563.602,Z 540.301,A 0.000,B 0.000,C 90.000,E1 270.229} C_DIS
LIN {X 0.271,Y -562.406,Z 540.292,A 0.000,B 0.000,C 90.000,E1 268.568} C_DIS
LIN {X 0.223,Y -561.480,Z 540.285,A 0.000,B 0.000,C 90.000,E1 267.192} C_DIS
LIN {X -0.275,Y -560.384,Z 540.275,A 0.000,B 0.000,C 90.000,E1 265.584} C_DIS
LIN {X 0.159,Y -559.564,Z 540.269,A 0.000,B 0.000,C 90.000,E1 264.432} C_DIS
LIN {X 0.229,Y -558.223,Z 540.260,A 0.000,B 0.000,C 90.000,E1 262.761} C_DIS
LIN {X 0.200,Y -557.107,Z 540.252,A 0.000,B 0.000,C 90.000,E1 261.376} C_DIS
LIN {X 0.057,Y -556.204,Z 540.248,A 0.000,B 0.000,C 90.000,E1 260.557} C_DIS
LIN {X -0.083,Y -553.505,Z 540.235,A 0.000,B 0.000,C 90.000,E1 258.342} C_DIS
LIN {X 0.107,Y -551.338,Z 540.226,A 0.000,B 0.000,C 90.000,E1 256.645} C_DIS
LIN {X 0.154,Y -549.781,Z 540.220,A 0.000,B 0.000,C 90.000,E1 255.519} C_DIS
LIN {X -0.251,Y -547.676,Z 540.212,A 0.000,B 0.000,C 90.000,E1 254.157} C_DIS
LIN {X -0.022,Y -545.337,Z 540.204,A 0.000,B 0.000,C 90.000,E1 252.725} C_DIS
LIN {X -0.189,Y -542.768,Z 540.196,A 0.000,B 0.000,C 90.000,E1 251.329} C_DIS
LIN {X 0.110,Y -540.070,Z 540.188,A 0.000,B 0.000,C 90.000,E1 249.880} C_DIS
LIN {X 0.254,Y -536.497,Z 540.179,A 0.000,B 0.000,C 90.000,E1 248.156} C_DIS
LIN {X 0.111,Y -533.333,Z 540.171,A 0.000,B 0.000,C 90.000,E1 246.741} C_DIS
LIN {X -0.076,Y -530.564,Z 540.165,A 0.000,B 0.000,C 90.000,E1 245.613} C_DIS
LIN {X -0.077,Y -527.659,Z 540.158,A 0.000,B 0.000,C 90.000,E1 244.460} C_DIS
LIN {X 0.045,Y -523.808,Z 540.150,A 0.000,B 0.000,C 90.000,E1 242.999} C_DIS
LIN {X -0.055,Y -520.620,Z 540.144,A 0.000,B 0.000,C 90.000,E1 241.847} C_DIS
LIN {X 0.073,Y -515.777,Z 540.134,A 0.000,B 0.000,C 90.000,E1 240.078} C_DIS
LIN {X -0.083,Y -512.389,Z 540.127,A 0.000,B 0.000,C 90.000,E1 238.918} C_DIS
LIN {X -0.212,Y -507.959,Z 540.119,A 0.000,B 0.000,C 90.000,E1 237.454} C_DIS
LIN {X 0.121,Y -503.524,Z 540.111,A 0.000,B 0.000,C 90.000,E1 235.928} C_DIS
LIN {X 0.248,Y -498.282,Z 540.101,A 0.000,B 0.000,C 90.000,E1 234.116} C_DIS
LIN {X -0.154,Y -493.228,Z 540.091,A 0.000,B 0.000,C 90.000,E1 232.351} C_DIS
LIN {X 0.089,Y -489.036,Z 540.082,A 0.000,B 0.000,C 90.000,E1 230.803} C_DIS
LIN {X -0.118,Y -484.982,Z 540.074,A 0.000,B 0.000,C 90.000,E1 229.299} C_DIS
LIN {X -0.276,Y -480.190,Z 540.064,A 0.000,B 0.000,C 90.000,E1 227.472} C_DIS
LIN {X -0.016,Y -474.018,Z 540.050,A 0.000,B 0.000,C 90.000,E1 224.960} C_DIS
LIN {X 0.128,Y -470.207,Z 540.041,A 0.000,B 0.000,C 90.000,E1 223.380} C_DIS
LIN {X -0.115,Y -466.576,Z 540.032,A 0.000,B 0.000,C 90.000,E1 221.838} C_DIS
LIN {X -0.071,Y -462.945,Z 540.024,A 0.000,B 0.000,C 90.000,E1 220.253} C_DIS
LIN {X -0.102,Y -459.373,Z 540.015,A 0.000,B 0.000,C 90.000,E1 218.669} C_DIS
LIN {X -0.038,Y -455.198,Z 540.004,A 0.000,B 0.000,C 90.000,E1 216.744} C_DIS
LIN {X -0.068,Y -451.154,Z 539.993,A 0.000,B 0.000,C 90.000,E1 214.818} C_DIS
LIN {X 0.214,Y -447.853,Z 539.984,A 0.000,B 0.000,C 90.000,E1 213.166} C_DIS
LIN {X -0.010,Y -442.818,Z 539.970,A 0.000,B 0.000,C 90.000,E1 210.590} C_DIS
LIN {X -0.071,Y -438.017,Z 539.955,A 0.000,B 0.000,C 90.000,E1 207.975} C_DIS
LIN {X -0.107,Y -434.095,Z 539.943,A 0.000,B 0.000,C 90.000,E1 205.668} C_DIS
LIN {X -0.063,Y -429.785,Z 539.928,A 0.000,B 0.000,C 90.000,E1 203.003} C_DIS
LIN {X 0.126,Y -426.765,Z 539.917,A 0.000,B 0.000,C 90.000,E1 200.972} C_DIS
LIN {X -0.064,Y -423.139,Z 539.902,A 0.000,B 0.000,C 90.000,E1 198.308} C_DIS
LIN {X 0.090,Y -420.559,Z 539.890,A 0.000,B 0.000,C 90.000,E1 196.260} C_DIS
LIN {X -0.108,Y -418.567,Z 539.881,A 0.000,B 0.000,C 90.000,E1 194.592} C_DIS
LIN {X -0.102,Y -416.892,Z 539.873,A 0.000,B 0.000,C 90.000,E1 193.231} C_DIS
LIN {X -0.169,Y -414.747,Z 539.864,A 0.000,B 0.000,C 90.000,E1 191.535} C_DIS
LIN {X 0.096,Y -412.325,Z 539.853,A 0.000,B 0.000,C 90.000,E1 189.443} C_DIS
LIN {X -0.134,Y -410.429,Z 539.843,A 0.000,B 0.000,C 90.000,E1 187.757} C_DIS
LIN {X -0.070,Y -407.967,Z 539.830,A 0.000,B 0.000,C 90.000,E1 185.334} C_DIS
LIN {X -0.151,Y -405.822,Z 539.816,A 0.000,B 0.000,C 90.000,E1 182.922} C_DIS
LIN {X 0.016,Y -403.422,Z 539.799,A 0.000,B 0.000,C 90.000,E1 179.771} C_DIS
LIN {X 0.079,Y -401.714,Z 539.779,A 0.000,B 0.000,C 90.000,E1 176.274} C_DIS
LIN {X -0.184,Y -400.916,Z 539.764,A 0.000,B 0.000,C 90.000,E1 173.514} C_DIS
LIN {X 0.055,Y -400.651,Z 539.746,A 0.000,B 0.000,C 90.000,E1 170.330} C_DIS
LIN {X 0.049,Y -400.836,Z 539.733,A 0.000,B 0.000,C 90.000,E1 167.881} C_DIS
LIN {X -0.087,Y -401.390,Z 539.717,A 0.000,B 0.000,C 90.000,E1 165.102} C_DIS
LIN {X -0.069,Y -402.246,Z 539.704,A 0.000,B 0.000,C 90.000,E1 162.653} C_DIS
LIN {X -0.009,Y -403.160,Z 539.692,A 0.000,B 0.000,C 90.000,E1 160.550} C_DIS
LIN {X -0.043,Y -404.301,Z 539.680,A 0.000,B 0.000,C 90.000,E1 158.465} C_DIS
LIN {X -0.175,Y -405.700,Z 539.667,A 0.000,B 0.000,C 90.000,E1 156.049} C_DIS
LIN {X -0.203,Y -406.643,Z 539.659,A 0.000,B 0.000,C 90.000,E1 154.665} C_DIS
LIN {X 0.142,Y -408.051,Z 539.648,A 0.000,B 0.000,C 90.000,E1 152.538} C_DIS
LIN {X -0.113,Y -409.175,Z 539.638,A 0.000,B 0.000,C 90.000,E1 150.845} C_DIS
LIN {X -0.071,Y -409.981,Z 539.630,A 0.000,B 0.000,C 90.000,E1 149.459} C_DIS
LIN {X -0.099,Y -410.769,Z 539.621,A 0.000,B 0.000,C 90.000,E1 147.740} C_DIS
LIN {X 0.051,Y -411.389,Z 539.613,A 0.000,B 0.000,C 90.000,E1 146.342} C_DIS
LIN {X 0.148,Y -411.955,Z 539.604,A 0.000,B 0.000,C 90.000,E1 144.609} C_DIS
LIN {X -0.087,Y -412.413,Z 539.594,A 0.000,B 0.000,C 90.000,E1 142.924} C_DIS
LIN {X 0.010,Y -412.685,Z 539.586,A 0.000,B 0.000,C 90.000,E1 141.537} C_DIS
LIN {X -0.036,Y -412.927,Z 539.577,A 0.000,B 0.000,C 90.000,E1 139.828} C_DIS
LIN {X 0.162,Y -413.052,Z 539.571,A 0.000,B 0.000,C 90.000,E1 138.771} C_DIS
LIN {X -0.055,Y -413.165,Z 539.560,A 0.000,B 0.000,C 90.000,E1 136.743} C_DIS
LIN {X -0.120,Y -413.252,Z 539.546,A 0.000,B 0.000,C 90.000,E1 134.352} C_DIS
LIN {X 0.083,Y -413.290,Z 539.537,A 0.000,B 0.000,C 90.000,E1 132.609} C_DIS
LIN {X -0.026,Y -413.253,Z 539.531,A 0.000,B 0.000,C 90.000,E1 131.595} C_DIS
LIN {X 0.030,Y -412.952,Z 539.523,A 0.000,B 0.000,C 90.000,E1 130.216} C_DIS
LIN {X -0.040,Y -412.592,Z 539.518,A 0.000,B 0.000,C 90.000,E1 129.197} C_DIS
LIN {X 0.059,Y -411.905,Z 539.510,A 0.000,B 0.000,C 90.000,E1 127.810} C_DIS
LIN {X 0.030,Y -411.601,Z 539.507,A 0.000,B 0.000,C 90.000,E1 127.282} C_DIS
LIN {X -0.008,Y -411.599,Z 539.507,A 0.000,B 0.000,C 90.000,E1 127.282} C_DIS
LIN {X 0.072,Y -415.133,Z 539.501,A 0.000,B 0.000,C 90.000,E1 126.091} C_DIS
LIN {X 0.003,Y -416.044,Z 539.499,A 0.000,B 0.000,C 90.000,E1 125.758} C_DIS
LIN {X 0.132,Y -425.558,Z 539.478,A 0.000,B 0.000,C 90.000,E1 122.005} C_DIS
LIN {X 0.076,Y -430.592,Z 539.469,A 0.000,B 0.000,C 90.000,E1 120.335} C_DIS
LIN {X 0.070,Y -441.500,Z 539.445,A 0.000,B 0.000,C 90.000,E1 116.027} C_DIS
LIN {X 0.197,Y -444.414,Z 539.439,A 0.000,B 0.000,C 90.000,E1 115.027} C_DIS
LIN {X 0.096,Y -445.897,Z 539.436,A 0.000,B 0.000,C 90.000,E1 114.387} C_DIS
LIN {X -0.183,Y -447.020,Z 539.433,A 0.000,B 0.000,C 90.000,E1 113.898} C_DIS
LIN {X -0.223,Y -447.063,Z 539.433,A 0.000,B 0.000,C 90.000,E1 113.898} C_DIS
LIN {X 0.148,Y -477.931,Z 539.426,A 0.000,B 0.000,C 90.000,E1 112.589} C_DIS
LIN {X -0.143,Y -488.290,Z 539.423,A 0.000,B 0.000,C 90.000,E1 112.206} C_DIS
LIN {X -0.173,Y -498.544,Z 539.421,A 0.000,B 0.000,C 90.000,E1 111.770} C_DIS
LIN {X 0.165,Y -508.757,Z 539.418,A 0.000,B 0.000,C 90.000,E1 111.280} C_DIS
LIN {X -0.051,Y -518.967,Z 539.416,A 0.000,B 0.000,C 90.000,E1 110.844} C_DIS
LIN {X -0.089,Y -528.737,Z 539.413,A 0.000,B 0.000,C 90.000,E1 110.375} C_DIS
LIN {X 0.047,Y -536.979,Z 539.411,A 0.000,B 0.000,C 90.000,E1 109.939} C_DIS
LIN {X -0.042,Y -544.983,Z 539.408,A 0.000,B 0.000,C 90.000,E1 109.504} C_DIS
LIN {X -0.233,Y -551.143,Z 539.406,A 0.000,B 0.000,C 90.000,E1 109.141} C_DIS
LIN {X 0.202,Y -556.667,Z 539.404,A 0.000,B 0.000,C 90.000,E1 108.725} C_DIS
LIN {X -0.288,Y -562.110,Z 539.402,A 0.000,B 0.000,C 90.000,E1 108.362} C_DIS
LIN {X 0.257,Y -567.248,Z 539.399,A 0.000,B 0.000,C 90.000,E1 107.873} C_DIS
LIN {X 0.144,Y -572.440,Z 539.397,A 0.000,B 0.000,C 90.000,E1 107.402} C_DIS
LIN {X 0.102,Y -578.300,Z 539.393,A 0.000,B 0.000,C 90.000,E1 106.804} C_DIS
LIN {X 0.120,Y -583.970,Z 539.390,A 0.000,B 0.000,C 90.000,E1 106.134} C_DIS
LIN {X 0.021,Y -588.295,Z 539.387,A 0.000,B 0.000,C 90.000,E1 105.607} C_DIS
LIN {X -0.122,Y -593.118,Z 539.383,A 0.000,B 0.000,C 90.000,E1 104.954} C_DIS
LIN {X -0.012,Y -600.096,Z 539.377,A 0.000,B 0.000,C 90.000,E1 103.883} C_DIS
LIN {X 0.252,Y -605.763,Z 539.372,A 0.000,B 0.000,C 90.000,E1 102.939} C_DIS
LIN {X -0.078,Y -610.441,Z 539.368,A 0.000,B 0.000,C 90.000,E1 102.187} C_DIS
LIN {X 0.130,Y -616.239,Z 539.362,A 0.000,B 0.000,C 90.000,E1 101.130} C_DIS
LIN {X 0.154,Y -620.088,Z 539.358,A 0.000,B 0.000,C 90.000,E1 100.366} C_DIS
LIN {X -0.251,Y -624.710,Z 539.352,A 0.000,B 0.000,C 90.000,E1 99.378} C_DIS
LIN {X 0.232,Y -628.186,Z 539.348,A 0.000,B 0.000,C 90.000,E1 98.568} C_DIS
